C03619=1061.195,-112.854,-61.247,171.285,25.780,154.842
C03620=1061.201,-112.604,-61.257,171.286,25.781,154.842
C03621=1061.207,-112.354,-61.267,171.288,25.782,154.842
C03622=1061.214,-112.105,-61.276,171.290,25.783,154.842
C03623=1061.219,-111.855,-61.286,171.292,25.784,154.841
C03624=1061.225,-111.605,-61.296,171.294,25.785,154.842
C03625=1061.232,-111.356,-61.306,171.296,25.786,154.841
C03626=1061.237,-111.107,-61.315,171.297,25.787,154.841
C03627=1061.243,-110.857,-61.325,171.299,25.788,154.841
C03628=1061.250,-110.606,-61.335,171.301,25.789,154.841
C03629=1061.256,-110.356,-61.344,171.303,25.790,154.841
C03630=1061.263,-110.107,-61.354,171.304,25.790,154.841
C03631=1061.268,-109.892,-61.363,171.306,25.792,154.841
C03632=1061.273,-109.677,-61.371,171.308,25.792,154.841
C03633=1061.279,-109.462,-61.380,171.310,25.793,154.841
C03634=1061.284,-109.247,-61.388,171.311,25.794,154.841
C03635=1061.289,-109.032,-61.396,171.312,25.795,154.841
C03636=1061.295,-108.817,-61.405,171.314,25.795,154.841
C03637=1061.300,-108.602,-61.414,171.316,25.797,154.841
C03638=1061.305,-108.387,-61.421,171.318,25.797,154.841
C03639=1061.311,-108.138,-61.432,171.320,25.798,154.841
C03640=1061.317,-107.888,-61.441,171.321,25.800,154.841
C03641=1061.323,-107.638,-61.451,171.323,25.800,154.841
C03642=1061.329,-107.388,-61.461,171.325,25.801,154.841
C03643=1061.335,-107.139,-61.471,171.327,25.803,154.841
C03644=1061.342,-106.888,-61.481,171.329,25.803,154.841
C03645=1061.348,-106.638,-61.491,171.330,25.804,154.841
C03646=1061.354,-106.388,-61.501,171.332,25.806,154.841
C03647=1061.360,-106.139,-61.511,171.334,25.807,154.841
C03648=1061.366,-105.889,-61.521,171.336,25.807,154.841
C03649=1061.373,-105.640,-61.530,171.337,25.809,154.841
C03650=1061.378,-105.390,-61.541,171.339,25.810,154.841
C03651=1061.384,-105.140,-61.551,171.341,25.811,154.841
C03652=1061.391,-104.890,-61.560,171.343,25.812,154.841
C03653=1061.396,-104.641,-61.571,171.344,25.813,154.841
C03654=1061.403,-104.391,-61.581,171.346,25.814,154.841
C03655=1061.409,-104.141,-61.590,171.348,25.815,154.841
C03656=1061.415,-103.892,-61.601,171.350,25.816,154.841
C03657=1061.421,-103.642,-61.611,171.352,25.817,154.841
C03658=1061.427,-103.393,-61.621,171.354,25.818,154.841
C03659=1061.434,-103.142,-61.631,171.356,25.820,154.841
C03660=1061.439,-102.892,-61.641,171.358,25.821,154.841
C03661=1061.446,-102.643,-61.651,171.359,25.822,154.841
C03662=1061.452,-102.393,-61.661,171.361,25.823,154.841
C03663=1061.458,-102.144,-61.672,171.363,25.824,154.841
C03664=1061.464,-101.894,-61.681,171.365,25.825,154.841
C03665=1061.470,-101.644,-61.691,171.366,25.826,154.841
C03666=1061.476,-101.395,-61.702,171.368,25.827,154.841
C03667=1061.483,-101.144,-61.712,171.370,25.828,154.841
C03668=1061.489,-100.895,-61.722,171.372,25.830,154.841
C03669=1061.494,-100.645,-61.732,171.373,25.831,154.841
C03670=1061.501,-100.396,-61.743,171.375,25.831,154.841
C03671=1061.507,-100.146,-61.752,171.377,25.833,154.841
C03672=1061.513,-99.896,-61.763,171.379,25.834,154.841
C03673=1061.519,-99.647,-61.773,171.380,25.835,154.841
C03674=1061.526,-99.397,-61.783,171.383,25.836,154.841
C03675=1061.535,-99.043,-61.798,171.385,25.838,154.841
C03676=1061.543,-98.690,-61.812,171.387,25.840,154.841
C03677=1061.552,-98.335,-61.827,171.390,25.841,154.841
C03678=1061.560,-97.982,-61.841,171.393,25.843,154.841
C03679=1061.567,-97.732,-61.851,171.394,25.844,154.841
C03680=1061.573,-97.483,-61.861,171.396,25.845,154.841
C03681=1061.579,-97.233,-61.872,171.398,25.846,154.841
C03682=1061.585,-96.982,-61.882,171.400,25.847,154.841
C03683=1061.591,-96.733,-61.893,171.401,25.849,154.841
C03684=1061.597,-96.484,-61.904,171.404,25.851,154.841
C03685=1061.603,-96.234,-61.913,171.406,25.852,154.841
C03686=1061.609,-95.984,-61.924,171.407,25.853,154.841
C03687=1061.615,-95.735,-61.934,171.409,25.854,154.841
C03688=1061.621,-95.485,-61.944,171.411,25.855,154.841
C03689=1061.627,-95.235,-61.956,171.413,25.857,154.841
C03690=1061.633,-94.985,-61.965,171.414,25.858,154.841
C03691=1061.639,-94.736,-61.976,171.416,25.859,154.841
C03692=1061.646,-94.486,-61.986,171.418,25.861,154.841
C03693=1061.651,-94.236,-61.997,171.419,25.862,154.841
C03694=1061.658,-93.986,-62.007,171.421,25.863,154.841
C03695=1061.664,-93.737,-62.018,171.423,25.864,154.841
C03696=1061.669,-93.487,-62.028,171.425,25.865,154.841
C03697=1061.676,-93.238,-62.039,171.426,25.867,154.841
C03698=1061.681,-92.988,-62.049,171.428,25.868,154.841
C03699=1061.689,-92.738,-62.060,171.430,25.870,154.841
C03700=1061.694,-92.488,-62.070,171.431,25.871,154.841
C03701=1061.700,-92.239,-62.081,171.433,25.872,154.841
C03702=1061.706,-91.990,-62.091,171.435,25.873,154.841
C03703=1061.712,-91.739,-62.102,171.438,25.875,154.842
C03704=1061.719,-91.490,-62.112,171.439,25.876,154.842
C03705=1061.724,-91.240,-62.123,171.441,25.878,154.842
C03706=1061.730,-90.991,-62.134,171.443,25.879,154.842
C03707=1061.737,-90.741,-62.145,171.444,25.880,154.842
C03708=1061.743,-90.491,-62.155,171.446,25.882,154.842
C03709=1061.748,-90.241,-62.166,171.448,25.883,154.842
C03710=1061.755,-89.992,-62.176,171.450,25.884,154.842
C03711=1061.761,-89.742,-62.187,171.451,25.885,154.842
C03712=1061.767,-89.492,-62.198,171.453,25.887,154.842
C03713=1061.773,-89.242,-62.208,171.455,25.888,154.842
C03714=1061.779,-88.992,-62.219,171.456,25.889,154.842
C03715=1061.786,-88.743,-62.229,171.458,25.891,154.842
C03716=1061.792,-88.494,-62.240,171.460,25.892,154.842
C03717=1061.797,-88.244,-62.251,171.461,25.894,154.842
C03718=1061.805,-87.994,-62.262,171.463,25.895,154.842
C03719=1061.810,-87.744,-62.272,171.465,25.896,154.842
C03720=1061.816,-87.495,-62.283,171.467,25.898,154.842
C03721=1061.823,-87.245,-62.293,171.469,25.899,154.842
C03722=1061.829,-86.995,-62.304,171.471,25.900,154.842
C03723=1061.834,-86.746,-62.315,171.473,25.902,154.843
C03724=1061.841,-86.496,-62.326,171.474,25.903,154.843
C03725=1061.847,-86.246,-62.337,171.476,25.904,154.843
C03726=1061.853,-85.997,-62.347,171.478,25.906,154.843
C03727=1061.860,-85.747,-62.358,171.479,25.907,154.843
C03728=1061.865,-85.497,-62.368,171.481,25.909,154.843
C03729=1061.872,-85.247,-62.379,171.483,25.910,154.843
C03730=1061.878,-84.998,-62.390,171.484,25.912,154.843
C03731=1061.884,-84.748,-62.401,171.486,25.913,154.843
C03732=1061.890,-84.498,-62.412,171.488,25.914,154.843
C03733=1061.896,-84.248,-62.423,171.490,25.916,154.843
C03734=1061.902,-83.999,-62.433,171.491,25.917,154.843
C03735=1061.909,-83.749,-62.444,171.493,25.919,154.843
C03736=1061.915,-83.499,-62.455,171.495,25.920,154.843
C03737=1061.922,-83.250,-62.466,171.497,25.922,154.843
C03738=1061.927,-83.000,-62.477,171.499,25.923,154.843
C03739=1061.935,-82.718,-62.489,171.501,25.924,154.843
C03740=1061.942,-82.436,-62.501,171.502,25.926,154.844
C03741=1061.948,-82.154,-62.514,171.505,25.928,154.844
C03742=1061.955,-81.872,-62.526,171.507,25.929,154.844
C03743=1061.961,-81.622,-62.537,171.508,25.931,154.844
C03744=1061.968,-81.372,-62.548,171.510,25.932,154.844
C03745=1061.974,-81.123,-62.559,171.512,25.933,154.844
C03746=1061.980,-80.873,-62.570,171.513,25.935,154.844
C03747=1061.987,-80.624,-62.580,171.515,25.936,154.844
C03748=1061.993,-80.373,-62.591,171.517,25.938,154.844
C03749=1061.999,-80.124,-62.602,171.518,25.939,154.844
C03750=1062.005,-79.874,-62.614,171.520,25.941,154.844
C03751=1062.011,-79.625,-62.625,171.522,25.942,154.844
C03752=1062.018,-79.376,-62.635,171.523,25.944,154.844
C03753=1062.024,-79.125,-62.647,171.526,25.945,154.844
C03754=1062.030,-78.876,-62.657,171.528,25.947,154.845
C03755=1062.036,-78.626,-62.669,171.529,25.949,154.845
C03756=1062.042,-78.376,-62.680,171.531,25.950,154.845
C03757=1062.048,-78.127,-62.692,171.533,25.952,154.845
C03758=1062.054,-77.877,-62.702,171.534,25.953,154.845
C03759=1062.060,-77.628,-62.713,171.536,25.955,154.845
C03760=1062.066,-77.378,-62.725,171.538,25.957,154.845
C03761=1062.072,-77.128,-62.735,171.539,25.958,154.845
C03762=1062.078,-76.878,-62.747,171.541,25.960,154.845
C03763=1062.084,-76.629,-62.758,171.543,25.961,154.845
C03764=1062.091,-76.379,-62.769,171.544,25.962,154.845
C03765=1062.096,-76.129,-62.780,171.546,25.964,154.846
C03766=1062.103,-75.879,-62.792,171.548,25.965,154.846
C03767=1062.109,-75.630,-62.803,171.549,25.967,154.846
C03768=1062.115,-75.380,-62.814,171.551,25.969,154.846
C03769=1062.121,-75.131,-62.825,171.553,25.970,154.846
C03770=1062.127,-74.880,-62.837,171.554,25.972,154.846
C03771=1062.133,-74.632,-62.848,171.557,25.974,154.846
C03772=1062.140,-74.382,-62.859,171.558,25.975,154.846
C03773=1062.146,-74.132,-62.870,171.560,25.977,154.846
C03774=1062.152,-73.882,-62.881,171.562,25.979,154.846
C03775=1062.158,-73.633,-62.893,171.563,25.980,154.847
C03776=1062.164,-73.383,-62.904,171.565,25.982,154.847
C03777=1062.170,-73.133,-62.915,171.567,25.983,154.847
C03778=1062.177,-72.884,-62.927,171.568,25.985,154.847
C03779=1062.182,-72.634,-62.938,171.570,25.987,154.847
C03780=1062.187,-72.384,-62.950,171.572,25.989,154.847
C03781=1062.194,-72.135,-62.962,171.573,25.990,154.847
C03782=1062.200,-71.885,-62.972,171.575,25.992,154.847
C03783=1062.206,-71.635,-62.984,171.577,25.993,154.848
C03784=1062.212,-71.386,-62.995,171.578,25.995,154.848
C03785=1062.218,-71.136,-63.007,171.580,25.997,154.848
C03786=1062.224,-70.887,-63.019,171.581,25.999,154.848
C03787=1062.230,-70.637,-63.030,171.583,26.000,154.848
C03788=1062.236,-70.387,-63.041,171.585,26.002,154.848
C03789=1062.242,-70.137,-63.053,171.586,26.003,154.848
C03790=1062.247,-69.888,-63.064,171.588,26.005,154.848
C03791=1062.254,-69.638,-63.076,171.590,26.007,154.849
C03792=1062.260,-69.389,-63.087,171.592,26.009,154.849
C03793=1062.266,-69.139,-63.099,171.594,26.011,154.849
C03794=1062.272,-68.889,-63.111,171.595,26.012,154.849
C03795=1062.278,-68.639,-63.122,171.597,26.014,154.849
C03796=1062.284,-68.389,-63.134,171.599,26.016,154.849
C03797=1062.290,-68.140,-63.145,171.600,26.018,154.849
C03798=1062.296,-67.890,-63.157,171.602,26.019,154.849
C03799=1062.302,-67.641,-63.168,171.603,26.021,154.850
C03800=1062.308,-67.391,-63.180,171.605,26.022,154.850
C03801=1062.314,-67.142,-63.191,171.607,26.024,154.850
C03802=1062.320,-66.892,-63.203,171.608,26.026,154.850
C03803=1062.327,-66.612,-63.216,171.610,26.028,154.850
C03804=1062.334,-66.332,-63.229,171.612,26.030,154.850
C03805=1062.340,-66.052,-63.242,171.614,26.032,154.850
C03806=1062.347,-65.772,-63.255,171.616,26.034,154.851
C03807=1062.354,-65.523,-63.267,171.617,26.036,154.851
C03808=1062.360,-65.273,-63.278,171.619,26.037,154.851
C03809=1062.366,-65.023,-63.290,171.621,26.039,154.851
C03810=1062.372,-64.773,-63.302,171.622,26.041,154.851
C03811=1062.378,-64.524,-63.313,171.624,26.043,154.851
C03812=1062.384,-64.274,-63.326,171.625,26.044,154.851
C03813=1062.390,-64.024,-63.337,171.627,26.046,154.852
C03814=1062.396,-63.775,-63.349,171.629,26.048,154.852
C03815=1062.403,-63.525,-63.360,171.631,26.050,154.852
C03816=1062.408,-63.276,-63.372,171.633,26.052,154.852
C03817=1062.415,-63.026,-63.384,171.634,26.053,154.852
C03818=1062.421,-62.776,-63.395,171.636,26.055,154.852
C03819=1062.426,-62.527,-63.408,171.638,26.057,154.852
C03820=1062.433,-62.277,-63.419,171.639,26.059,154.852
C03821=1062.439,-62.027,-63.431,171.641,26.060,154.853
C03822=1062.445,-61.778,-63.442,171.643,26.062,154.853
C03823=1062.451,-61.529,-63.455,171.644,26.064,154.853
C03824=1062.458,-61.278,-63.466,171.646,26.066,154.853
C03825=1062.464,-61.029,-63.478,171.647,26.067,154.853
C03826=1062.470,-60.780,-63.490,171.649,26.069,154.853
C03827=1062.476,-60.529,-63.501,171.651,26.071,154.853
C03828=1062.483,-60.280,-63.513,171.652,26.073,154.854
C03829=1062.488,-60.031,-63.526,171.654,26.074,154.854
C03830=1062.494,-59.781,-63.538,171.656,26.076,154.854
C03831=1062.501,-59.531,-63.549,171.657,26.078,154.854
C03832=1062.506,-59.282,-63.561,171.659,26.080,154.854
C03833=1062.513,-59.032,-63.573,171.660,26.082,154.854
C03834=1062.519,-58.782,-63.584,171.662,26.084,154.855
C03835=1062.525,-58.532,-63.597,171.664,26.086,154.855
C03836=1062.531,-58.283,-63.608,171.665,26.087,154.855
C03837=1062.538,-58.034,-63.620,171.667,26.089,154.855
C03838=1062.544,-57.784,-63.633,171.669,26.091,154.855
C03839=1062.550,-57.534,-63.644,171.671,26.093,154.855
C03840=1062.556,-57.285,-63.656,171.673,26.095,154.855
C03841=1062.562,-57.035,-63.668,171.674,26.096,154.856
C03842=1062.569,-56.785,-63.680,171.676,26.098,154.856
C03843=1062.574,-56.535,-63.693,171.677,26.100,154.856
C03844=1062.581,-56.286,-63.705,171.679,26.102,154.856
C03845=1062.587,-56.036,-63.716,171.681,26.104,154.856
C03846=1062.593,-55.786,-63.728,171.682,26.106,154.856
C03847=1062.599,-55.537,-63.740,171.684,26.107,154.857
C03848=1062.606,-55.287,-63.752,171.685,26.109,154.857
C03849=1062.612,-55.037,-63.765,171.687,26.111,154.857
C03850=1062.618,-54.788,-63.776,171.689,26.113,154.857
C03851=1062.624,-54.539,-63.789,171.690,26.115,154.857
C03852=1062.630,-54.288,-63.800,171.692,26.117,154.857
C03853=1062.637,-54.039,-63.812,171.693,26.119,154.858
C03854=1062.643,-53.789,-63.825,171.695,26.120,154.858
C03855=1062.649,-53.540,-63.836,171.697,26.122,154.858
C03856=1062.656,-53.290,-63.848,171.698,26.124,154.858
C03857=1062.661,-53.041,-63.861,171.700,26.126,154.858
C03858=1062.668,-52.791,-63.873,171.701,26.128,154.858
C03859=1062.674,-52.541,-63.885,171.703,26.130,154.858
C03860=1062.681,-52.292,-63.897,171.705,26.131,154.859
C03861=1062.687,-52.042,-63.910,171.706,26.133,154.859
C03862=1062.693,-51.793,-63.921,171.708,26.135,154.859
C03863=1062.699,-51.543,-63.933,171.710,26.137,154.859
C03864=1062.705,-51.293,-63.946,171.711,26.139,154.859
C03865=1062.712,-51.044,-63.958,171.714,26.141,154.859
C03866=1062.718,-50.794,-63.970,171.715,26.143,154.860
C03867=1062.725,-50.516,-63.983,171.717,26.145,154.860
C03868=1062.732,-50.237,-63.997,171.718,26.147,154.860
C03869=1062.738,-49.958,-64.011,171.720,26.149,154.860
C03870=1062.745,-49.679,-64.025,171.722,26.151,154.860
C03871=1062.751,-49.430,-64.037,171.724,26.154,154.861
C03872=1062.757,-49.180,-64.049,171.726,26.155,154.861
C03873=1062.763,-48.930,-64.062,171.727,26.158,154.861
C03874=1062.769,-48.681,-64.074,171.729,26.159,154.861
C03875=1062.776,-48.432,-64.087,171.730,26.161,154.861
C03876=1062.782,-48.182,-64.099,171.732,26.164,154.862
C03877=1062.787,-47.933,-64.112,171.733,26.165,154.862
C03878=1062.794,-47.683,-64.123,171.735,26.168,154.862
C03879=1062.800,-47.433,-64.136,171.737,26.169,154.862
C03880=1062.806,-47.183,-64.149,171.738,26.172,154.862
C03881=1062.812,-46.933,-64.161,171.740,26.173,154.863
C03882=1062.818,-46.684,-64.173,171.741,26.175,154.863
C03883=1062.824,-46.435,-64.186,171.743,26.178,154.863
C03884=1062.830,-46.185,-64.199,171.744,26.179,154.863
C03885=1062.836,-45.935,-64.211,171.746,26.182,154.863
C03886=1062.842,-45.686,-64.223,171.748,26.183,154.863
C03887=1062.848,-45.436,-64.236,171.749,26.186,154.864
C03888=1062.854,-45.186,-64.248,171.751,26.187,154.864
C03889=1062.860,-44.937,-64.261,171.752,26.189,154.864
C03890=1062.867,-44.687,-64.273,171.754,26.191,154.864
C03891=1062.873,-44.437,-64.286,171.755,26.193,154.864
C03892=1062.879,-44.188,-64.299,171.757,26.196,154.865
C03893=1062.884,-43.938,-64.311,171.759,26.197,154.865
C03894=1062.891,-43.689,-64.323,171.760,26.200,154.865
C03895=1062.897,-43.440,-64.336,171.762,26.201,154.865
C03896=1062.903,-43.190,-64.348,171.763,26.204,154.866
C03897=1062.909,-42.940,-64.361,171.765,26.205,154.866
C03898=1062.916,-42.691,-64.374,171.766,26.208,154.866
C03899=1062.922,-42.441,-64.386,171.768,26.210,154.866
C03900=1062.928,-42.191,-64.399,171.770,26.212,154.866
C03901=1062.934,-41.942,-64.412,171.771,26.214,154.866
C03902=1062.940,-41.692,-64.424,171.773,26.216,154.867
C03903=1062.946,-41.442,-64.437,171.774,26.218,154.867
C03904=1062.953,-41.193,-64.450,171.776,26.220,154.867
C03905=1062.958,-40.943,-64.462,171.777,26.222,154.867
C03906=1062.964,-40.693,-64.475,171.779,26.224,154.868
C03907=1062.971,-40.444,-64.487,171.781,26.226,154.868
C03908=1062.977,-40.194,-64.500,171.782,26.228,154.868
C03909=1062.983,-39.945,-64.513,171.784,26.230,154.868
C03910=1062.989,-39.695,-64.526,171.785,26.232,154.868
C03911=1062.995,-39.445,-64.539,171.788,26.234,154.868
C03912=1063.002,-39.196,-64.551,171.789,26.237,154.869
C03913=1063.008,-38.947,-64.564,171.791,26.238,154.869
C03914=1063.014,-38.697,-64.576,171.792,26.241,154.869
C03915=1063.020,-38.447,-64.589,171.794,26.243,154.869
C03916=1063.026,-38.198,-64.602,171.796,26.245,154.870
C03917=1063.032,-37.948,-64.615,171.797,26.247,154.870
C03918=1063.038,-37.698,-64.628,171.799,26.249,154.870
C03919=1063.044,-37.449,-64.641,171.800,26.251,154.870
C03920=1063.050,-37.199,-64.654,171.802,26.253,154.871
C03921=1063.056,-36.949,-64.666,171.803,26.256,154.871
C03922=1063.062,-36.699,-64.679,171.805,26.257,154.871
C03923=1063.068,-36.450,-64.692,171.806,26.260,154.871
C03924=1063.074,-36.200,-64.705,171.808,26.262,154.871
C03925=1063.081,-35.951,-64.718,171.810,26.264,154.872
C03926=1063.086,-35.701,-64.731,171.811,26.266,154.872
C03927=1063.093,-35.452,-64.744,171.813,26.269,154.872
C03928=1063.099,-35.202,-64.756,171.814,26.270,154.872
C03929=1063.105,-34.953,-64.770,171.816,26.273,154.873
C03930=1063.111,-34.703,-64.782,171.817,26.275,154.873
C03931=1063.117,-34.425,-64.797,171.819,26.277,154.873
C03932=1063.124,-34.146,-64.812,171.820,26.280,154.873
C03933=1063.131,-33.869,-64.826,171.822,26.282,154.874
C03934=1063.138,-33.591,-64.840,171.824,26.284,154.874
C03935=1063.143,-33.341,-64.853,171.826,26.286,154.874
C03936=1063.150,-33.092,-64.866,171.827,26.289,154.874
C03937=1063.156,-32.842,-64.880,171.829,26.291,154.874
C03938=1063.162,-32.592,-64.892,171.830,26.293,154.875
C03939=1063.169,-32.342,-64.906,171.832,26.295,154.875
C03940=1063.174,-32.093,-64.918,171.834,26.297,154.875
C03941=1063.181,-31.843,-64.932,171.835,26.300,154.875
C03942=1063.187,-31.594,-64.945,171.837,26.302,154.876
C03943=1063.193,-31.344,-64.957,171.838,26.304,154.876
C03944=1063.199,-31.095,-64.971,171.840,26.306,154.876
C03945=1063.205,-30.846,-64.984,171.841,26.308,154.876
C03946=1063.210,-30.595,-64.997,171.843,26.310,154.877
C03947=1063.217,-30.346,-65.010,171.844,26.312,154.877
C03948=1063.223,-30.096,-65.023,171.846,26.315,154.877
C03949=1063.229,-29.846,-65.037,171.847,26.317,154.877
C03950=1063.236,-29.597,-65.050,171.849,26.319,154.877
C03951=1063.242,-29.348,-65.063,171.851,26.321,154.878
C03952=1063.248,-29.098,-65.076,171.852,26.323,154.878
C03953=1063.254,-28.849,-65.089,171.854,26.326,154.878
C03954=1063.260,-28.599,-65.102,171.855,26.327,154.878
C03955=1063.267,-28.349,-65.115,171.857,26.330,154.879
C03956=1063.273,-28.100,-65.128,171.858,26.332,154.879
C03957=1063.279,-27.850,-65.142,171.860,26.334,154.879
C03958=1063.285,-27.601,-65.155,171.861,26.337,154.879
C03959=1063.290,-27.351,-65.168,171.863,26.338,154.880
C03960=1063.297,-27.102,-65.181,171.864,26.341,154.880
C03961=1063.303,-26.852,-65.195,171.866,26.343,154.880
C03962=1063.310,-26.602,-65.208,171.867,26.345,154.880
C03963=1063.316,-26.352,-65.221,171.869,26.348,154.881
C03964=1063.321,-26.103,-65.235,171.870,26.350,154.881
C03965=1063.327,-25.854,-65.248,171.872,26.352,154.881
C03966=1063.333,-25.604,-65.261,171.874,26.354,154.881
C03967=1063.339,-25.355,-65.275,171.875,26.356,154.882
C03968=1063.345,-25.105,-65.288,171.877,26.359,154.882
C03969=1063.352,-24.855,-65.301,171.878,26.361,154.882
C03970=1063.357,-24.605,-65.315,171.880,26.363,154.882
C03971=1063.363,-24.356,-65.328,171.881,26.366,154.883
C03972=1063.370,-24.107,-65.342,171.882,26.368,154.883
C03973=1063.375,-23.857,-65.355,171.883,26.370,154.883
C03974=1063.381,-23.607,-65.368,171.885,26.372,154.884
C03975=1063.388,-23.357,-65.382,171.886,26.375,154.884
C03976=1063.393,-23.108,-65.396,171.888,26.377,154.884
C03977=1063.399,-22.859,-65.409,171.889,26.379,154.884
C03978=1063.406,-22.609,-65.422,171.891,26.382,154.885
C03979=1063.411,-22.360,-65.436,171.893,26.383,154.885
C03980=1063.418,-22.110,-65.450,171.894,26.386,154.885
C03981=1063.424,-21.860,-65.463,171.896,26.388,154.885
C03982=1063.430,-21.611,-65.477,171.897,26.390,154.886
C03983=1063.436,-21.362,-65.490,171.899,26.393,154.886
C03984=1063.442,-21.112,-65.503,171.900,26.395,154.886
C03985=1063.448,-20.862,-65.517,171.902,26.397,154.886
C03986=1063.454,-20.613,-65.531,171.903,26.399,154.887
C03987=1063.461,-20.364,-65.544,171.905,26.402,154.887
C03988=1063.466,-20.113,-65.557,171.906,26.404,154.887
C03989=1063.473,-19.863,-65.571,171.908,26.406,154.887
C03990=1063.479,-19.614,-65.584,171.909,26.409,154.888
C03991=1063.484,-19.365,-65.598,171.911,26.411,154.888
C03992=1063.491,-19.115,-65.611,171.912,26.413,154.888
C03993=1063.497,-18.865,-65.625,171.914,26.416,154.888
C03994=1063.503,-18.616,-65.639,171.915,26.418,154.889
C03995=1063.510,-18.337,-65.654,171.917,26.420,154.889
C03996=1063.516,-18.058,-65.669,171.919,26.423,154.889
C03997=1063.524,-17.779,-65.684,171.921,26.426,154.890
C03998=1063.530,-17.500,-65.700,171.922,26.428,154.890
C03999=1063.536,-17.250,-65.713,171.924,26.430,154.890
C04000=1063.543,-17.001,-65.727,171.925,26.433,154.890
C04001=1063.549,-16.752,-65.741,171.927,26.435,154.891
C04002=1063.555,-16.502,-65.755,171.928,26.437,154.891
C04003=1063.562,-16.252,-65.769,171.930,26.440,154.891
C04004=1063.567,-16.003,-65.782,171.931,26.442,154.892
C04005=1063.573,-15.754,-65.796,171.933,26.444,154.892
C04006=1063.580,-15.504,-65.809,171.935,26.447,154.892
C04007=1063.586,-15.254,-65.823,171.936,26.449,154.892
C04008=1063.592,-15.005,-65.836,171.938,26.451,154.893
C04009=1063.597,-14.755,-65.850,171.939,26.453,154.893
C04010=1063.604,-14.506,-65.865,171.941,26.456,154.893
C04011=1063.610,-14.256,-65.879,171.942,26.458,154.893
C04012=1063.615,-14.007,-65.892,171.944,26.460,154.894
C04013=1063.622,-13.757,-65.906,171.945,26.463,154.894
C04014=1063.628,-13.507,-65.920,171.947,26.466,154.894
C04015=1063.634,-13.258,-65.934,171.948,26.468,154.895
C04016=1063.640,-13.008,-65.948,171.950,26.470,154.895
C04017=1063.646,-12.759,-65.962,171.950,26.472,154.895
C04018=1063.652,-12.509,-65.975,171.952,26.475,154.895
C04019=1063.658,-12.259,-65.989,171.953,26.477,154.896
C04020=1063.664,-12.010,-66.004,171.955,26.479,154.896
C04021=1063.670,-11.761,-66.017,171.956,26.482,154.896
C04022=1063.676,-11.511,-66.032,171.958,26.484,154.897
C04023=1063.682,-11.261,-66.045,171.959,26.487,154.897
C04024=1063.688,-11.012,-66.059,171.961,26.489,154.897
C04025=1063.694,-10.762,-66.074,171.962,26.491,154.897
C04026=1063.700,-10.513,-66.087,171.964,26.494,154.898
C04027=1063.706,-10.264,-66.102,171.965,26.496,154.898
C04028=1063.712,-10.014,-66.116,171.967,26.499,154.898
C04029=1063.718,-9.764,-66.129,171.968,26.501,154.899
C04030=1063.724,-9.515,-66.143,171.970,26.503,154.899
C04031=1063.730,-9.265,-66.158,171.971,26.506,154.899
C04032=1063.737,-9.016,-66.171,171.973,26.508,154.899
C04033=1063.743,-8.766,-66.185,171.974,26.510,154.900
C04034=1063.749,-8.517,-66.199,171.976,26.513,154.900
C04035=1063.755,-8.267,-66.213,171.977,26.515,154.900
C04036=1063.761,-8.017,-66.227,171.979,26.518,154.901
C04037=1063.767,-7.768,-66.241,171.980,26.520,154.901
C04038=1063.773,-7.518,-66.256,171.982,26.522,154.901
C04039=1063.779,-7.269,-66.270,171.984,26.525,154.901
C04040=1063.785,-7.020,-66.283,171.985,26.527,154.902
C04041=1063.791,-6.770,-66.298,171.986,26.530,154.902
C04042=1063.797,-6.521,-66.312,171.988,26.532,154.902
C04043=1063.804,-6.271,-66.326,171.990,26.534,154.903
C04044=1063.810,-6.022,-66.340,171.990,26.537,154.903
C04045=1063.816,-5.771,-66.355,171.992,26.539,154.903
C04046=1063.821,-5.522,-66.369,171.993,26.541,154.903
C04047=1063.828,-5.273,-66.383,171.995,26.544,154.904
C04048=1063.834,-5.023,-66.397,171.996,26.546,154.904
C04049=1063.840,-4.773,-66.412,171.998,26.549,154.904
C04050=1063.846,-4.524,-66.425,171.999,26.551,154.905
C04051=1063.853,-4.274,-66.440,172.001,26.553,154.905
C04052=1063.858,-4.025,-66.454,172.002,26.556,154.905
C04053=1063.865,-3.776,-66.468,172.004,26.558,154.906
C04054=1063.871,-3.526,-66.482,172.005,26.561,154.906
C04055=1063.877,-3.277,-66.497,172.007,26.563,154.906
C04056=1063.883,-3.027,-66.511,172.008,26.565,154.906
C04057=1063.889,-2.778,-66.525,172.010,26.568,154.907
C04058=1063.895,-2.527,-66.540,172.011,26.570,154.907
C04059=1063.901,-2.248,-66.556,172.013,26.573,154.907
C04060=1063.908,-1.967,-66.571,172.014,26.576,154.908
C04061=1063.915,-1.686,-66.589,172.016,26.579,154.908
C04062=1063.921,-1.406,-66.605,172.018,26.582,154.908
C04063=1063.927,-1.156,-66.619,172.020,26.584,154.909
C04064=1063.933,-0.907,-66.633,172.021,26.587,154.909
C04065=1063.939,-0.656,-66.648,172.022,26.589,154.909
C04066=1063.945,-0.408,-66.662,172.023,26.591,154.910
C04067=1063.951,-0.158,-66.677,172.025,26.594,154.910
C04068=1063.957,0.092,-66.691,172.026,26.596,154.910
C04069=1063.963,0.341,-66.706,172.027,26.599,154.911
C04070=1063.969,0.590,-66.721,172.029,26.602,154.911
C04071=1063.975,0.840,-66.734,172.031,26.604,154.911
C04072=1063.981,1.090,-66.749,172.032,26.607,154.912
C04073=1063.987,1.339,-66.764,172.034,26.609,154.912
C04074=1063.993,1.589,-66.778,172.035,26.611,154.912
C04075=1063.999,1.838,-66.793,172.036,26.614,154.913
C04076=1064.005,2.087,-66.808,172.038,26.616,154.913
C04077=1064.011,2.338,-66.822,172.040,26.619,154.913
C04078=1064.017,2.587,-66.837,172.041,26.622,154.914
C04079=1064.023,2.836,-66.851,172.043,26.624,154.914
C04080=1064.029,3.086,-66.865,172.044,26.626,154.914
C04081=1064.035,3.336,-66.880,172.045,26.629,154.914
C04082=1064.041,3.584,-66.895,172.047,26.631,154.915
C04083=1064.047,3.834,-66.910,172.047,26.634,154.915
C04084=1064.053,4.084,-66.924,172.049,26.636,154.915
C04085=1064.059,4.333,-66.939,172.051,26.639,154.916
C04086=1064.065,4.582,-66.953,172.052,26.641,154.916
C04087=1064.071,4.832,-66.968,172.054,26.644,154.916
C04088=1064.077,5.082,-66.982,172.055,26.646,154.917
C04089=1064.083,5.331,-66.997,172.057,26.649,154.917
C04090=1064.089,5.581,-67.012,172.058,26.651,154.917
C04091=1064.095,5.830,-67.026,172.060,26.653,154.918
C04092=1064.102,6.079,-67.041,172.061,26.656,154.918
C04093=1064.107,6.329,-67.055,172.063,26.659,154.918
C04094=1064.113,6.579,-67.070,172.064,26.662,154.919
C04095=1064.120,6.828,-67.085,172.066,26.664,154.919
C04096=1064.126,7.077,-67.100,172.067,26.666,154.919
C04097=1064.132,7.327,-67.115,172.068,26.669,154.920
C04098=1064.138,7.576,-67.129,172.070,26.671,154.920
C04099=1064.144,7.826,-67.144,172.071,26.673,154.920
C04100=1064.150,8.076,-67.158,172.072,26.676,154.920
C04101=1064.156,8.325,-67.173,172.074,26.678,154.921
C04102=1064.162,8.574,-67.188,172.075,26.681,154.921
C04103=1064.169,8.824,-67.203,172.077,26.684,154.921
C04104=1064.174,9.073,-67.218,172.078,26.686,154.922
C04105=1064.180,9.323,-67.233,172.080,26.689,154.922
C04106=1064.186,9.572,-67.248,172.081,26.691,154.922
C04107=1064.192,9.822,-67.263,172.083,26.693,154.923
C04108=1064.199,10.072,-67.277,172.084,26.696,154.923
C04109=1064.204,10.321,-67.291,172.086,26.699,154.923
C04110=1064.211,10.571,-67.306,172.087,26.701,154.924
C04111=1064.217,10.820,-67.321,172.089,26.704,154.924
C04112=1064.223,11.070,-67.336,172.090,26.706,154.924
C04113=1064.229,11.319,-67.351,172.092,26.709,154.925
C04114=1064.236,11.569,-67.366,172.093,26.711,154.925
C04115=1064.242,11.818,-67.381,172.094,26.713,154.925
C04116=1064.247,12.067,-67.396,172.095,26.716,154.926
C04117=1064.253,12.317,-67.411,172.097,26.718,154.926
C04118=1064.260,12.567,-67.426,172.098,26.721,154.926
C04119=1064.266,12.816,-67.440,172.100,26.723,154.927
C04120=1064.272,13.065,-67.455,172.101,26.726,154.927
C04121=1064.278,13.315,-67.470,172.103,26.729,154.927
C04122=1064.285,13.565,-67.485,172.104,26.731,154.927
C04123=1064.292,13.847,-67.502,172.106,26.734,154.928
C04124=1064.299,14.130,-67.519,172.107,26.737,154.928
C04125=1064.305,14.412,-67.536,172.109,26.740,154.929
C04126=1064.312,14.694,-67.553,172.111,26.743,154.929
C04127=1064.318,14.944,-67.568,172.112,26.745,154.929
C04128=1064.324,15.194,-67.583,172.114,26.748,154.930
C04129=1064.330,15.442,-67.599,172.115,26.750,154.930
C04130=1064.336,15.692,-67.614,172.116,26.753,154.930
C04131=1064.342,15.942,-67.629,172.117,26.755,154.931
C04132=1064.348,16.192,-67.644,172.119,26.758,154.931
C04133=1064.354,16.440,-67.659,172.120,26.760,154.931
C04134=1064.360,16.690,-67.674,172.122,26.763,154.932
C04135=1064.366,16.940,-67.689,172.123,26.765,154.932
C04136=1064.372,17.188,-67.705,172.125,26.768,154.932
C04137=1064.378,17.438,-67.720,172.126,26.770,154.933
C04138=1064.384,17.688,-67.735,172.128,26.773,154.933
C04139=1064.391,17.938,-67.750,172.129,26.776,154.933
C04140=1064.396,18.187,-67.765,172.131,26.778,154.934
C04141=1064.402,18.437,-67.780,172.132,26.781,154.934
C04142=1064.409,18.686,-67.796,172.134,26.784,154.934
C04143=1064.414,18.936,-67.811,172.134,26.786,154.935
C04144=1064.420,19.185,-67.826,172.136,26.788,154.935
C04145=1064.426,19.434,-67.841,172.137,26.791,154.935
C04146=1064.432,19.684,-67.857,172.139,26.794,154.936
C04147=1064.439,19.933,-67.872,172.140,26.796,154.936
C04148=1064.445,20.183,-67.887,172.142,26.799,154.936
C04149=1064.450,20.432,-67.902,172.143,26.801,154.937
C04150=1064.457,20.681,-67.918,172.145,26.804,154.937
C04151=1064.463,20.931,-67.933,172.146,26.806,154.937
C04152=1064.469,21.181,-67.948,172.148,26.809,154.938
C04153=1064.474,21.430,-67.963,172.149,26.812,154.938
C04154=1064.481,21.679,-67.979,172.151,26.814,154.938
C04155=1064.486,21.929,-67.995,172.152,26.817,154.939
C04156=1064.493,22.179,-68.010,172.153,26.819,154.939
C04157=1064.498,22.427,-68.026,172.154,26.822,154.939
C04158=1064.504,22.677,-68.040,172.156,26.824,154.940
C04159=1064.510,22.927,-68.056,172.157,26.827,154.940
C04160=1064.517,23.176,-68.072,172.159,26.829,154.940
C04161=1064.522,23.426,-68.087,172.160,26.832,154.941
C04162=1064.528,23.675,-68.102,172.162,26.835,154.941
C04163=1064.534,23.924,-68.118,172.163,26.837,154.941
C04164=1064.541,24.174,-68.133,172.165,26.840,154.942
C04165=1064.547,24.423,-68.149,172.166,26.842,154.942
C04166=1064.553,24.673,-68.164,172.168,26.845,154.942
C04167=1064.559,24.923,-68.180,172.169,26.848,154.943
C04168=1064.565,25.171,-68.195,172.171,26.850,154.943
C04169=1064.570,25.421,-68.211,172.171,26.853,154.944
C04170=1064.577,25.670,-68.226,172.173,26.855,154.944
C04171=1064.583,25.920,-68.242,172.174,26.858,154.944
C04172=1064.589,26.169,-68.257,172.176,26.860,154.945
C04173=1064.595,26.419,-68.273,172.177,26.863,154.945
C04174=1064.601,26.669,-68.288,172.179,26.866,154.945
C04175=1064.607,26.918,-68.304,172.180,26.868,154.946
C04176=1064.613,27.167,-68.319,172.182,26.871,154.946
C04177=1064.619,27.417,-68.335,172.183,26.873,154.946
C04178=1064.625,27.666,-68.350,172.185,26.876,154.947
C04179=1064.631,27.916,-68.366,172.186,26.879,154.947
C04180=1064.637,28.166,-68.382,172.188,26.881,154.947
C04181=1064.644,28.415,-68.397,172.188,26.883,154.948
C04182=1064.649,28.665,-68.413,172.190,26.886,154.948
C04183=1064.655,28.913,-68.428,172.191,26.889,154.948
C04184=1064.661,29.163,-68.444,172.193,26.891,154.949
C04185=1064.667,29.412,-68.460,172.194,26.894,154.949
C04186=1064.673,29.662,-68.476,172.196,26.897,154.949
C04187=1064.680,29.946,-68.494,172.197,26.900,154.950
C04188=1064.687,30.229,-68.511,172.199,26.903,154.950
C04189=1064.694,30.513,-68.529,172.201,26.906,154.951
C04190=1064.700,30.797,-68.548,172.202,26.909,154.951
C04191=1064.707,31.047,-68.563,172.204,26.912,154.951
C04192=1064.713,31.296,-68.579,172.205,26.915,154.952
C04193=1064.718,31.545,-68.595,172.206,26.917,154.952
C04194=1064.724,31.795,-68.611,172.207,26.919,154.952
C04195=1064.730,32.044,-68.626,172.209,26.922,154.953
C04196=1064.736,32.294,-68.642,172.210,26.925,154.953
C04197=1064.742,32.543,-68.658,172.212,26.927,154.954
C04198=1064.748,32.793,-68.674,172.213,26.930,154.954
C04199=1064.754,33.042,-68.689,172.215,26.932,154.954
C04200=1064.760,33.292,-68.705,172.216,26.935,154.955
C04201=1064.766,33.541,-68.722,172.218,26.938,154.955
C04202=1064.772,33.791,-68.737,172.219,26.940,154.955
C04203=1064.778,34.040,-68.753,172.221,26.943,154.956
C04204=1064.784,34.289,-68.769,172.222,26.946,154.956
C04205=1064.790,34.539,-68.785,172.223,26.948,154.956
C04206=1064.796,34.789,-68.801,172.224,26.951,154.957
C04207=1064.803,35.038,-68.817,172.226,26.953,154.957
C04208=1064.809,35.287,-68.833,172.227,26.956,154.957
C04209=1064.814,35.536,-68.848,172.229,26.959,154.958
C04210=1064.820,35.786,-68.864,172.230,26.961,154.958
C04211=1064.826,36.035,-68.880,172.232,26.964,154.958
C04212=1064.832,36.284,-68.896,172.233,26.967,154.959
C04213=1064.838,36.533,-68.913,172.235,26.969,154.959
C04214=1064.844,36.783,-68.928,172.236,26.972,154.960
C04215=1064.850,37.033,-68.944,172.238,26.974,154.960
C04216=1064.857,37.282,-68.960,172.239,26.977,154.960
C04217=1064.862,37.531,-68.976,172.240,26.980,154.961
C04218=1064.868,37.780,-68.992,172.241,26.982,154.961
C04219=1064.874,38.030,-69.008,172.243,26.985,154.961
C04220=1064.880,38.280,-69.024,172.244,26.988,154.962
C04221=1064.886,38.529,-69.041,172.246,26.991,154.962
C04222=1064.892,38.778,-69.057,172.247,26.993,154.962
C04223=1064.898,39.028,-69.073,172.249,26.996,154.963
C04224=1064.904,39.277,-69.089,172.250,26.999,154.963
C04225=1064.909,39.527,-69.105,172.252,27.001,154.964
C04226=1064.915,39.776,-69.121,172.253,27.004,154.964
C04227=1064.921,40.026,-69.137,172.255,27.006,154.964
C04228=1064.928,40.275,-69.153,172.256,27.009,154.965
C04229=1064.934,40.524,-69.169,172.257,27.011,154.965
C04230=1064.940,40.774,-69.186,172.258,27.014,154.965
C04231=1064.946,41.023,-69.202,172.260,27.017,154.966
C04232=1064.952,41.272,-69.218,172.261,27.020,154.966
C04233=1064.958,41.522,-69.234,172.263,27.022,154.966
C04234=1064.964,41.771,-69.251,172.264,27.025,154.967
C04235=1064.970,42.021,-69.267,172.266,27.028,154.967
C04236=1064.976,42.270,-69.283,172.267,27.030,154.967
C04237=1064.982,42.520,-69.300,172.269,27.033,154.968
C04238=1064.988,42.769,-69.316,172.270,27.036,154.968
C04239=1064.994,43.018,-69.332,172.272,27.039,154.969
C04240=1065.000,43.268,-69.348,172.272,27.041,154.969
C04241=1065.006,43.517,-69.365,172.274,27.043,154.969
C04242=1065.012,43.766,-69.381,172.275,27.046,154.970
C04243=1065.017,44.016,-69.398,172.277,27.049,154.970
C04244=1065.023,44.265,-69.414,172.278,27.051,154.970
C04245=1065.029,44.515,-69.430,172.280,27.054,154.971
C04246=1065.035,44.764,-69.447,172.281,27.057,154.971
C04247=1065.041,45.013,-69.463,172.283,27.060,154.972
C04248=1065.046,45.263,-69.480,172.284,27.063,154.972
C04249=1065.052,45.512,-69.496,172.286,27.066,154.972
C04250=1065.058,45.762,-69.512,172.287,27.068,154.973
C04251=1065.065,46.046,-69.531,172.288,27.071,154.973
C04252=1065.071,46.330,-69.550,172.290,27.074,154.974
C04253=1065.078,46.614,-69.569,172.291,27.077,154.974
C04254=1065.085,46.898,-69.587,172.293,27.080,154.974
C04255=1065.091,47.147,-69.604,172.294,27.083,154.975
C04256=1065.097,47.396,-69.621,172.296,27.086,154.975
C04257=1065.103,47.645,-69.637,172.297,27.088,154.976
C04258=1065.109,47.895,-69.653,172.299,27.091,154.976
C04259=1065.114,48.144,-69.670,172.300,27.094,154.976
C04260=1065.120,48.394,-69.686,172.302,27.097,154.977
C04261=1065.126,48.642,-69.703,172.303,27.100,154.977
C04262=1065.132,48.892,-69.720,172.305,27.102,154.977
C04263=1065.137,49.141,-69.736,172.305,27.104,154.978
C04264=1065.144,49.392,-69.753,172.307,27.107,154.978
C04265=1065.150,49.641,-69.769,172.308,27.110,154.979
C04266=1065.156,49.890,-69.785,172.310,27.113,154.979
C04267=1065.161,50.139,-69.803,172.311,27.115,154.979
C04268=1065.167,50.389,-69.819,172.313,27.118,154.980
C04269=1065.173,50.638,-69.836,172.314,27.121,154.980
C04270=1065.179,50.887,-69.852,172.316,27.124,154.980
C04271=1065.184,51.136,-69.869,172.317,27.127,154.981
C04272=1065.191,51.386,-69.886,172.319,27.129,154.981
C04273=1065.197,51.636,-69.902,172.320,27.132,154.982
C04274=1065.203,51.885,-69.919,172.322,27.134,154.982
C04275=1065.208,52.134,-69.936,172.322,27.137,154.982
C04276=1065.214,52.383,-69.952,172.324,27.140,154.983
C04277=1065.220,52.633,-69.969,172.325,27.142,154.983
C04278=1065.226,52.883,-69.987,172.327,27.145,154.983
C04279=1065.232,53.132,-70.003,172.328,27.148,154.984
C04280=1065.238,53.381,-70.019,172.330,27.151,154.984
C04281=1065.245,53.630,-70.036,172.331,27.153,154.985
C04282=1065.250,53.880,-70.053,172.333,27.156,154.985
C04283=1065.256,54.130,-70.070,172.334,27.159,154.985
C04284=1065.263,54.378,-70.086,172.336,27.161,154.986
C04285=1065.268,54.628,-70.103,172.337,27.164,154.986
C04286=1065.274,54.877,-70.120,172.339,27.166,154.986
C04287=1065.280,55.126,-70.137,172.339,27.169,154.987
C04288=1065.286,55.377,-70.154,172.341,27.172,154.987
C04289=1065.292,55.625,-70.171,172.342,27.175,154.988
C04290=1065.298,55.875,-70.187,172.344,27.178,154.988
C04291=1065.304,56.124,-70.203,172.345,27.180,154.988
C04292=1065.310,56.374,-70.221,172.347,27.183,154.989
C04293=1065.316,56.623,-70.237,172.348,27.185,154.989
C04294=1065.322,56.872,-70.254,172.350,27.188,154.989
C04295=1065.328,57.121,-70.271,172.351,27.191,154.990
C04296=1065.334,57.371,-70.289,172.353,27.193,154.990
C04297=1065.340,57.620,-70.305,172.354,27.196,154.991
C04298=1065.346,57.870,-70.322,172.356,27.199,154.991
C04299=1065.352,58.119,-70.339,172.356,27.201,154.991
C04300=1065.358,58.369,-70.355,172.358,27.204,154.992
C04301=1065.364,58.618,-70.373,172.359,27.207,154.992
C04302=1065.370,58.867,-70.389,172.361,27.209,154.992
C04303=1065.377,59.116,-70.406,172.362,27.212,154.993
C04304=1065.382,59.366,-70.423,172.364,27.215,154.993
C04305=1065.388,59.615,-70.440,172.365,27.217,154.993
C04306=1065.393,59.865,-70.457,172.367,27.220,154.994
C04307=1065.400,60.114,-70.474,172.368,27.222,154.994
C04308=1065.406,60.363,-70.491,172.370,27.225,154.995
C04309=1065.412,60.612,-70.508,172.371,27.228,154.995
C04310=1065.419,60.862,-70.526,172.373,27.230,154.995
C04311=1065.425,61.111,-70.542,172.374,27.233,154.996
C04312=1065.430,61.360,-70.559,172.376,27.236,154.996
C04313=1065.437,61.610,-70.576,172.376,27.239,154.996
C04314=1065.443,61.859,-70.593,172.378,27.241,154.997
C04315=1065.450,62.143,-70.612,172.380,27.244,154.997
C04316=1065.457,62.426,-70.632,172.382,27.247,154.998
C04317=1065.463,62.710,-70.651,172.383,27.250,154.998
C04318=1065.470,62.993,-70.670,172.385,27.253,154.998
C04319=1065.476,63.243,-70.688,172.386,27.256,154.999
C04320=1065.482,63.492,-70.705,172.388,27.259,154.999
C04321=1065.488,63.742,-70.723,172.389,27.261,154.999
C04322=1065.495,63.991,-70.740,172.391,27.264,155.000
C04323=1065.501,64.240,-70.756,172.392,27.267,155.000
C04324=1065.507,64.490,-70.774,172.394,27.269,155.001
C04325=1065.513,64.739,-70.791,172.395,27.272,155.001
C04326=1065.518,64.988,-70.808,172.397,27.274,155.001
C04327=1065.524,65.238,-70.825,172.398,27.277,155.002
C04328=1065.531,65.487,-70.842,172.399,27.280,155.002
C04329=1065.536,65.736,-70.860,172.400,27.283,155.003
C04330=1065.543,65.986,-70.877,172.402,27.285,155.003
C04331=1065.548,66.235,-70.894,172.403,27.288,155.003
C04332=1065.554,66.485,-70.912,172.405,27.290,155.004
C04333=1065.560,66.734,-70.928,172.406,27.293,155.004
C04334=1065.566,66.983,-70.946,172.408,27.296,155.004
C04335=1065.572,67.233,-70.964,172.409,27.299,155.005
C04336=1065.578,67.481,-70.981,172.411,27.302,155.005
C04337=1065.584,67.730,-70.998,172.412,27.304,155.006
C04338=1065.589,67.981,-71.016,172.414,27.307,155.006
C04339=1065.596,68.230,-71.033,172.415,27.310,155.006
C04340=1065.602,68.479,-71.051,172.417,27.312,155.007
C04341=1065.607,68.728,-71.068,172.418,27.315,155.007
C04342=1065.614,68.977,-71.085,172.419,27.317,155.007
C04343=1065.620,69.227,-71.103,172.420,27.320,155.008
C04344=1065.625,69.476,-71.120,172.422,27.323,155.008
C04345=1065.632,69.726,-71.137,172.423,27.326,155.009
C04346=1065.637,69.975,-71.155,172.425,27.329,155.009
C04347=1065.643,70.224,-71.172,172.426,27.331,155.009
C04348=1065.649,70.474,-71.190,172.428,27.334,155.010
C04349=1065.655,70.722,-71.207,172.429,27.336,155.010
C04350=1065.661,70.972,-71.225,172.431,27.339,155.010
C04351=1065.667,71.221,-71.243,172.432,27.342,155.011
C04352=1065.672,71.471,-71.260,172.434,27.345,155.011
C04353=1065.678,71.721,-71.278,172.435,27.348,155.012
C04354=1065.684,71.969,-71.294,172.437,27.351,155.012
C04355=1065.691,72.219,-71.312,172.438,27.353,155.012
C04356=1065.696,72.468,-71.330,172.440,27.356,155.013
C04357=1065.702,72.717,-71.348,172.441,27.358,155.013
C04358=1065.708,72.967,-71.365,172.442,27.361,155.014
C04359=1065.714,73.216,-71.382,172.444,27.364,155.014
C04360=1065.720,73.465,-71.400,172.445,27.367,155.014
C04361=1065.726,73.714,-71.418,172.446,27.369,155.015
C04362=1065.732,73.964,-71.436,172.448,27.372,155.015
C04363=1065.737,74.213,-71.453,172.450,27.374,155.015
C04364=1065.743,74.463,-71.471,172.451,27.377,155.016
C04365=1065.750,74.712,-71.488,172.453,27.380,155.016
C04366=1065.755,74.961,-71.506,172.454,27.383,155.017
C04367=1065.761,75.210,-71.524,172.456,27.386,155.017
C04368=1065.767,75.460,-71.541,172.457,27.389,155.017
C04369=1065.773,75.709,-71.559,172.459,27.391,155.018
C04370=1065.778,75.958,-71.577,172.460,27.394,155.018
C04371=1065.784,76.208,-71.595,172.462,27.396,155.019
C04372=1065.791,76.457,-71.612,172.463,27.399,155.019
C04373=1065.797,76.706,-71.630,172.464,27.402,155.019
C04374=1065.803,76.955,-71.648,172.465,27.405,155.020
C04375=1065.809,77.205,-71.666,172.467,27.407,155.020
C04376=1065.814,77.454,-71.684,172.468,27.410,155.020
C04377=1065.820,77.703,-71.701,172.470,27.412,155.021
C04378=1065.826,77.953,-71.719,172.471,27.415,155.021
C04379=1065.834,78.236,-71.739,172.473,27.418,155.022
C04380=1065.840,78.520,-71.759,172.475,27.422,155.022
C04381=1065.846,78.803,-71.780,172.477,27.425,155.023
C04382=1065.853,79.086,-71.800,172.478,27.428,155.023
C04383=1065.859,79.336,-71.818,172.479,27.431,155.023
C04384=1065.864,79.585,-71.836,172.481,27.433,155.024
C04385=1065.870,79.835,-71.854,172.483,27.436,155.024
C04386=1065.876,80.083,-71.872,172.484,27.439,155.025
C04387=1065.882,80.333,-71.890,172.486,27.441,155.025
C04388=1065.888,80.582,-71.908,172.487,27.444,155.025
C04389=1065.894,80.832,-71.926,172.489,27.447,155.026
C04390=1065.900,81.080,-71.944,172.490,27.450,155.026
C04391=1065.906,81.330,-71.962,172.492,27.453,155.026
C04392=1065.911,81.579,-71.980,172.493,27.455,155.027
C04393=1065.917,81.829,-71.998,172.494,27.458,155.027
C04394=1065.923,82.077,-72.016,172.495,27.461,155.028
C04395=1065.929,82.327,-72.034,172.497,27.463,155.028
C04396=1065.935,82.577,-72.052,172.498,27.466,155.028
C04397=1065.940,82.826,-72.070,172.500,27.469,155.029
C04398=1065.947,83.075,-72.089,172.501,27.471,155.029
C04399=1065.952,83.324,-72.106,172.503,27.474,155.030
C04400=1065.958,83.574,-72.124,172.504,27.477,155.030
C04401=1065.964,83.823,-72.142,172.506,27.480,155.030
C04402=1065.970,84.072,-72.160,172.507,27.483,155.031
C04403=1065.976,84.321,-72.178,172.509,27.485,155.031
C04404=1065.982,84.571,-72.197,172.510,27.488,155.031
C04405=1065.988,84.820,-72.215,172.512,27.491,155.032
C04406=1065.993,85.070,-72.233,172.513,27.493,155.032
C04407=1066.000,85.319,-72.251,172.515,27.496,155.033
C04408=1066.005,85.568,-72.269,172.516,27.499,155.033
C04409=1066.012,85.817,-72.287,172.518,27.502,155.033
C04410=1066.018,86.067,-72.305,172.519,27.505,155.034
C04411=1066.022,86.316,-72.324,172.521,27.507,155.034
C04412=1066.029,86.565,-72.342,172.522,27.510,155.035
C04413=1066.035,86.815,-72.360,172.524,27.512,155.035
C04414=1066.041,87.063,-72.378,172.525,27.515,155.035
C04415=1066.047,87.313,-72.396,172.527,27.518,155.036
C04416=1066.053,87.561,-72.415,172.528,27.521,155.036
C04417=1066.058,87.811,-72.433,172.529,27.523,155.037
C04418=1066.065,88.061,-72.452,172.531,27.526,155.037
C04419=1066.070,88.310,-72.469,172.532,27.528,155.037
C04420=1066.076,88.559,-72.487,172.534,27.531,155.038
C04421=1066.083,88.808,-72.506,172.535,27.534,155.038
C04422=1066.088,89.057,-72.523,172.537,27.537,155.038
C04423=1066.094,89.307,-72.543,172.538,27.540,155.039
C04424=1066.100,89.557,-72.561,172.540,27.542,155.039
C04425=1066.106,89.805,-72.579,172.541,27.545,155.040
C04426=1066.112,90.054,-72.598,172.543,27.547,155.040
C04427=1066.118,90.304,-72.616,172.544,27.550,155.040
C04428=1066.124,90.553,-72.635,172.546,27.553,155.041
C04429=1066.130,90.802,-72.652,172.547,27.556,155.041
C04430=1066.136,91.052,-72.671,172.549,27.558,155.041
C04431=1066.141,91.302,-72.690,172.550,27.561,155.042
C04432=1066.147,91.550,-72.708,172.552,27.564,155.042
C04433=1066.153,91.800,-72.726,172.553,27.566,155.043
C04434=1066.159,92.049,-72.745,172.555,27.569,155.043
C04435=1066.165,92.298,-72.763,172.557,27.572,155.043
C04436=1066.170,92.548,-72.782,172.558,27.575,155.044
C04437=1066.177,92.797,-72.800,172.560,27.578,155.044
C04438=1066.182,93.045,-72.819,172.561,27.580,155.045
C04439=1066.188,93.295,-72.837,172.563,27.583,155.045
C04440=1066.194,93.544,-72.856,172.564,27.586,155.045
C04441=1066.199,93.793,-72.875,172.566,27.589,155.046
C04442=1066.205,94.043,-72.893,172.567,27.592,155.046
C04443=1066.212,94.325,-72.914,172.569,27.594,155.047
C04444=1066.219,94.609,-72.935,172.570,27.597,155.047
C04445=1066.225,94.893,-72.956,172.572,27.601,155.048
C04446=1066.232,95.177,-72.977,172.574,27.604,155.048
C04447=1066.238,95.426,-72.996,172.576,27.606,155.048
C04448=1066.243,95.675,-73.015,172.577,27.609,155.049
C04449=1066.250,95.924,-73.034,172.579,27.612,155.049
C04450=1066.256,96.174,-73.051,172.580,27.615,155.050
C04451=1066.261,96.423,-73.071,172.582,27.618,155.050
C04452=1066.267,96.672,-73.089,172.583,27.620,155.050
C04453=1066.273,96.921,-73.108,172.585,27.623,155.051
C04454=1066.279,97.171,-73.126,172.586,27.625,155.051
C04455=1066.285,97.420,-73.145,172.588,27.628,155.051
C04456=1066.291,97.669,-73.164,172.589,27.631,155.052
C04457=1066.296,97.918,-73.183,172.591,27.634,155.052
C04458=1066.303,98.167,-73.202,172.592,27.637,155.053
C04459=1066.308,98.417,-73.220,172.594,27.639,155.053
C04460=1066.315,98.666,-73.239,172.595,27.642,155.053
C04461=1066.320,98.915,-73.258,172.597,27.644,155.054
C04462=1066.326,99.164,-73.276,172.598,27.647,155.054
C04463=1066.332,99.414,-73.296,172.600,27.650,155.055
C04464=1066.338,99.663,-73.314,172.601,27.653,155.055
C04465=1066.344,99.912,-73.332,172.603,27.656,155.055
C04466=1066.349,100.161,-73.351,172.605,27.658,155.056
C04467=1066.356,100.410,-73.370,172.606,27.661,155.056
C04468=1066.361,100.660,-73.389,172.608,27.663,155.056
C04469=1066.368,100.909,-73.408,172.609,27.666,155.057
C04470=1066.374,101.158,-73.427,172.611,27.669,155.057
C04471=1066.379,101.407,-73.446,172.612,27.672,155.058
C04472=1066.385,101.656,-73.464,172.614,27.675,155.058
C04473=1066.391,101.906,-73.484,172.615,27.677,155.058
C04474=1066.396,102.155,-73.503,172.617,27.680,155.059
C04475=1066.403,102.404,-73.521,172.618,27.683,155.059
C04476=1066.408,102.653,-73.540,172.620,27.686,155.060
C04477=1066.414,102.902,-73.560,172.621,27.689,155.060
C04478=1066.419,103.152,-73.579,172.623,27.691,155.060
C04479=1066.426,103.401,-73.597,172.624,27.694,155.061
C04480=1066.431,103.650,-73.617,172.626,27.697,155.061
C04481=1066.437,103.899,-73.636,172.627,27.699,155.062
C04482=1066.443,104.148,-73.654,172.629,27.702,155.062
C04483=1066.449,104.398,-73.673,172.631,27.705,155.062
C04484=1066.454,104.647,-73.693,172.632,27.707,155.063
C04485=1066.460,104.896,-73.712,172.634,27.710,155.063
C04486=1066.466,105.146,-73.731,172.635,27.713,155.064
C04487=1066.472,105.394,-73.749,172.637,27.716,155.064
C04488=1066.477,105.644,-73.769,172.638,27.719,155.064
C04489=1066.483,105.893,-73.788,172.640,27.721,155.065
C04490=1066.489,106.142,-73.807,172.641,27.724,155.065
C04491=1066.495,106.392,-73.826,172.643,27.727,155.066
C04492=1066.501,106.641,-73.845,172.644,27.729,155.066
C04493=1066.507,106.890,-73.864,172.646,27.732,155.066
C04494=1066.513,107.139,-73.884,172.647,27.735,155.067
C04495=1066.518,107.388,-73.903,172.649,27.738,155.067
C04496=1066.524,107.637,-73.922,172.650,27.740,155.067
C04497=1066.530,107.886,-73.940,172.652,27.743,155.068
C04498=1066.536,108.136,-73.960,172.654,27.746,155.068
C04499=1066.542,108.385,-73.979,172.655,27.749,155.069
C04500=1066.548,108.634,-73.999,172.657,27.751,155.069
C04501=1066.553,108.883,-74.018,172.658,27.754,155.069
C04502=1066.560,109.133,-74.037,172.660,27.756,155.070
C04503=1066.566,109.382,-74.056,172.661,27.759,155.070
C04504=1066.571,109.631,-74.075,172.663,27.762,155.071
C04505=1066.577,109.880,-74.095,172.664,27.765,155.071
C04506=1066.584,110.129,-74.114,172.666,27.768,155.071
C04507=1066.590,110.412,-74.136,172.667,27.770,155.072
C04508=1066.596,110.697,-74.157,172.670,27.774,155.072
C04509=1066.603,110.980,-74.179,172.671,27.777,155.073
C04510=1066.610,111.264,-74.202,172.673,27.780,155.073
C04511=1066.615,111.513,-74.221,172.674,27.782,155.073
C04512=1066.621,111.762,-74.241,172.676,27.785,155.074
C04513=1066.627,112.011,-74.260,172.677,27.788,155.074
C04514=1066.633,112.260,-74.279,172.679,27.791,155.075
C04515=1066.639,112.509,-74.299,172.680,27.793,155.075
C04516=1066.645,112.759,-74.318,172.683,27.797,155.075
C04517=1066.651,113.008,-74.337,172.684,27.799,155.076
C04518=1066.657,113.257,-74.357,172.686,27.802,155.076
C04519=1066.663,113.506,-74.376,172.688,27.804,155.077
C04520=1066.668,113.756,-74.395,172.689,27.807,155.077
C04521=1066.674,114.005,-74.415,172.691,27.810,155.077
C04522=1066.680,114.254,-74.435,172.692,27.813,155.078
C04523=1066.686,114.503,-74.454,172.694,27.815,155.078
C04524=1066.691,114.752,-74.474,172.695,27.818,155.079
C04525=1066.697,115.001,-74.493,172.697,27.821,155.079
C04526=1066.703,115.250,-74.513,172.698,27.824,155.079
C04527=1066.708,115.499,-74.532,172.700,27.827,155.080
C04528=1066.714,115.748,-74.553,172.701,27.829,155.080
C04529=1066.719,115.998,-74.572,172.703,27.832,155.081
C04530=1066.725,116.247,-74.591,172.704,27.835,155.081
C04531=1066.731,116.496,-74.611,172.706,27.838,155.081
C04532=1066.737,116.745,-74.630,172.708,27.840,155.082
C04533=1066.743,116.994,-74.650,172.709,27.843,155.082
C04534=1066.748,117.244,-74.669,172.711,27.846,155.083
C04535=1066.754,117.493,-74.690,172.712,27.849,155.083
C04536=1066.759,117.742,-74.709,172.714,27.852,155.083
C04537=1066.765,117.991,-74.729,172.715,27.854,155.084
C04538=1066.771,118.240,-74.748,172.718,27.857,155.084
C04539=1066.777,118.489,-74.768,172.719,27.860,155.085
C04540=1066.783,118.739,-74.788,172.721,27.863,155.085
C04541=1066.788,118.988,-74.808,172.722,27.866,155.085
C04542=1066.794,119.237,-74.828,172.724,27.868,155.086
C04543=1066.800,119.486,-74.847,172.725,27.871,155.086
C04544=1066.806,119.735,-74.867,172.727,27.874,155.087
C04545=1066.811,119.984,-74.887,172.728,27.877,155.087
C04546=1066.817,120.233,-74.907,172.730,27.880,155.087
C04547=1066.822,120.483,-74.926,172.732,27.882,155.088
C04548=1066.828,120.732,-74.946,172.733,27.885,155.088
C04549=1066.834,120.981,-74.966,172.735,27.887,155.088
C04550=1066.840,121.230,-74.986,172.736,27.890,155.089
C04551=1066.845,121.479,-75.006,172.738,27.893,155.089
C04552=1066.851,121.728,-75.026,172.739,27.896,155.090
C04553=1066.857,121.978,-75.046,172.742,27.899,155.090
C04554=1066.863,122.227,-75.066,172.743,27.901,155.090
C04555=1066.869,122.476,-75.086,172.745,27.904,155.091
C04556=1066.874,122.725,-75.105,172.746,27.907,155.091
C04557=1066.880,122.974,-75.125,172.748,27.910,155.092
C04558=1066.886,123.223,-75.145,172.750,27.912,155.092
C04559=1066.892,123.472,-75.165,172.751,27.915,155.092
C04560=1066.898,123.721,-75.185,172.753,27.918,155.093
C04561=1066.903,123.970,-75.205,172.754,27.921,155.093
C04562=1066.909,124.219,-75.225,172.756,27.923,155.094
C04563=1066.916,124.469,-75.245,172.757,27.926,155.094
C04564=1066.922,124.718,-75.265,172.759,27.929,155.094
C04565=1066.927,124.967,-75.285,172.761,27.932,155.095
C04566=1066.933,125.216,-75.305,172.763,27.934,155.095
C04567=1066.939,125.466,-75.324,172.764,27.937,155.096
C04568=1066.945,125.714,-75.344,172.766,27.940,155.096
C04569=1066.950,125.963,-75.365,172.768,27.943,155.096
C04570=1066.956,126.213,-75.385,172.769,27.945,155.097
C04571=1066.963,126.497,-75.408,172.771,27.948,155.097
C04572=1066.970,126.780,-75.431,172.773,27.951,155.098
C04573=1066.976,127.063,-75.453,172.775,27.955,155.098
C04574=1066.983,127.346,-75.476,172.777,27.958,155.098
C04575=1066.988,127.595,-75.497,172.779,27.960,155.099
C04576=1066.994,127.844,-75.516,172.780,27.963,155.099
C04577=1067.000,128.094,-75.536,172.782,27.966,155.100
C04578=1067.007,128.343,-75.556,172.783,27.969,155.100
C04579=1067.012,128.592,-75.577,172.785,27.971,155.100
C04580=1067.018,128.841,-75.597,172.786,27.974,155.101
C04581=1067.024,129.090,-75.617,172.788,27.976,155.101
C04582=1067.030,129.340,-75.637,172.790,27.979,155.102
C04583=1067.036,129.589,-75.657,172.792,27.982,155.102
C04584=1067.042,129.837,-75.677,172.794,27.985,155.102
C04585=1067.048,130.086,-75.697,172.795,27.988,155.103
C04586=1067.054,130.336,-75.718,172.797,27.990,155.103
C04587=1067.060,130.585,-75.738,172.798,27.993,155.103
C04588=1067.066,130.834,-75.758,172.800,27.995,155.104
C04589=1067.071,131.083,-75.778,172.801,27.998,155.104
C04590=1067.077,131.333,-75.798,172.803,28.001,155.105
C04591=1067.083,131.582,-75.818,172.805,28.004,155.105
C04592=1067.088,131.831,-75.839,172.807,28.006,155.105
C04593=1067.094,132.080,-75.859,172.809,28.009,155.106
C04594=1067.100,132.330,-75.880,172.810,28.012,155.106
C04595=1067.107,132.578,-75.900,172.812,28.014,155.107
C04596=1067.112,132.827,-75.921,172.813,28.017,155.107
C04597=1067.118,133.076,-75.941,172.815,28.020,155.107
C04598=1067.123,133.325,-75.961,172.816,28.023,155.108
C04599=1067.130,133.574,-75.982,172.819,28.026,155.108
C04600=1067.135,133.823,-76.002,172.820,28.029,155.109
C04601=1067.141,134.072,-76.022,172.822,28.031,155.109
C04602=1067.146,134.321,-76.043,172.824,28.034,155.109
C04603=1067.152,134.571,-76.064,172.825,28.037,155.110
C04604=1067.158,134.820,-76.084,172.827,28.040,155.110
C04605=1067.163,135.069,-76.104,172.828,28.042,155.111
C04606=1067.170,135.317,-76.125,172.831,28.045,155.111
C04607=1067.175,135.567,-76.146,172.832,28.048,155.111
C04608=1067.181,135.816,-76.166,172.834,28.050,155.112
C04609=1067.187,136.065,-76.186,172.835,28.053,155.112
C04610=1067.193,136.315,-76.207,172.837,28.056,155.112
C04611=1067.199,136.564,-76.227,172.839,28.059,155.113
C04612=1067.204,136.812,-76.249,172.840,28.061,155.113
C04613=1067.210,137.061,-76.268,172.843,28.064,155.114
C04614=1067.216,137.311,-76.289,172.844,28.067,155.114
C04615=1067.222,137.560,-76.309,172.846,28.070,155.114
C04616=1067.227,137.809,-76.330,172.847,28.073,155.115
C04617=1067.233,138.058,-76.352,172.849,28.075,155.115
C04618=1067.239,138.307,-76.371,172.850,28.078,155.116
C04619=1067.245,138.556,-76.392,172.852,28.081,155.116
C04620=1067.251,138.805,-76.414,172.855,28.084,155.116
C04621=1067.257,139.054,-76.434,172.856,28.086,155.117
C04622=1067.262,139.303,-76.454,172.858,28.089,155.117
C04623=1067.268,139.553,-76.475,172.859,28.092,155.118
C04624=1067.274,139.801,-76.496,172.861,28.094,155.118
C04625=1067.279,140.050,-76.516,172.862,28.097,155.118
C04626=1067.285,140.300,-76.537,172.865,28.100,155.119
C04627=1067.291,140.549,-76.559,172.866,28.103,155.119
C04628=1067.297,140.797,-76.578,172.868,28.106,155.120
C04629=1067.303,141.047,-76.599,172.870,28.108,155.120
C04630=1067.308,141.296,-76.621,172.871,28.111,155.120
C04631=1067.314,141.545,-76.641,172.873,28.114,155.121
C04632=1067.320,141.794,-76.663,172.875,28.117,155.121
C04633=1067.326,142.043,-76.683,172.877,28.120,155.122
C04634=1067.331,142.292,-76.703,172.878,28.122,155.122
C04635=1067.338,142.575,-76.728,172.880,28.125,155.122
C04636=1067.344,142.859,-76.752,172.882,28.129,155.123
C04637=1067.351,143.142,-76.775,172.884,28.131,155.123
C04638=1067.357,143.425,-76.798,172.886,28.135,155.124
C04639=1067.363,143.674,-76.820,172.888,28.138,155.124
C04640=1067.368,143.923,-76.841,172.889,28.141,155.125
C04641=1067.375,144.173,-76.862,172.891,28.143,155.125
C04642=1067.380,144.422,-76.883,172.894,28.146,155.125
C04643=1067.386,144.670,-76.903,172.895,28.149,155.126
C04644=1067.392,144.920,-76.924,172.897,28.152,155.126
C04645=1067.398,145.168,-76.946,172.898,28.155,155.127
C04646=1067.403,145.418,-76.967,172.900,28.157,155.127
C04647=1067.409,145.667,-76.988,172.902,28.160,155.127
C04648=1067.415,145.916,-77.009,172.904,28.162,155.128
C04649=1067.421,146.165,-77.029,172.905,28.165,155.128
C04650=1067.426,146.414,-77.050,172.907,28.168,155.128
C04651=1067.433,146.663,-77.072,172.909,28.171,155.129
C04652=1067.438,146.911,-77.093,172.911,28.174,155.129
C04653=1067.444,147.161,-77.114,172.913,28.176,155.130
C04654=1067.450,147.410,-77.135,172.914,28.179,155.130
C04655=1067.455,147.660,-77.156,172.916,28.182,155.130
C04656=1067.461,147.908,-77.177,172.918,28.185,155.131
C04657=1067.467,148.157,-77.199,172.920,28.188,155.131
C04658=1067.473,148.406,-77.219,172.921,28.190,155.132
C04659=1067.479,148.655,-77.241,172.923,28.193,155.132
C04660=1067.485,148.904,-77.261,172.925,28.196,155.132
C04661=1067.491,149.154,-77.283,172.927,28.199,155.133
C04662=1067.496,149.402,-77.304,172.929,28.202,155.133
C04663=1067.501,149.651,-77.326,172.930,28.204,155.134
C04664=1067.507,149.901,-77.347,172.932,28.207,155.134
C04665=1067.513,150.149,-77.368,172.933,28.210,155.134
C04666=1067.519,150.399,-77.390,172.936,28.213,155.135
C04667=1067.524,150.648,-77.410,172.938,28.216,155.135
C04668=1067.530,150.897,-77.432,172.939,28.218,155.136
C04669=1067.536,151.145,-77.453,172.941,28.221,155.136
C04670=1067.542,151.395,-77.475,172.943,28.224,155.136
C04671=1067.547,151.644,-77.495,172.945,28.227,155.137
C04672=1067.553,151.893,-77.517,172.946,28.230,155.137
C04673=1067.559,152.141,-77.538,172.948,28.232,155.138
C04674=1067.565,152.391,-77.560,172.950,28.235,155.138
C04675=1067.571,152.639,-77.581,172.952,28.238,155.138
C04676=1067.576,152.889,-77.602,172.954,28.241,155.139
C04677=1067.581,153.138,-77.624,172.955,28.244,155.139
C04678=1067.587,153.387,-77.646,172.958,28.247,155.140
C04679=1067.593,153.635,-77.667,172.959,28.249,155.140
C04680=1067.599,153.885,-77.688,172.961,28.252,155.140
C04681=1067.605,154.134,-77.710,172.962,28.255,155.141
C04682=1067.611,154.383,-77.731,172.965,28.258,155.141
C04683=1067.617,154.632,-77.752,172.966,28.261,155.142
C04684=1067.622,154.881,-77.774,172.968,28.263,155.142
C04685=1067.628,155.130,-77.795,172.970,28.265,155.142
C04686=1067.633,155.379,-77.817,172.972,28.268,155.143
C04687=1067.639,155.628,-77.839,172.974,28.271,155.143
C04688=1067.645,155.876,-77.860,172.975,28.274,155.144
C04689=1067.651,156.126,-77.882,172.977,28.277,155.144
C04690=1067.657,156.375,-77.904,172.979,28.280,155.144
C04691=1067.662,156.624,-77.925,172.981,28.283,155.145
C04692=1067.668,156.873,-77.947,172.983,28.286,155.145
C04693=1067.674,157.121,-77.968,172.984,28.288,155.146
C04694=1067.679,157.371,-77.990,172.987,28.291,155.146
C04695=1067.685,157.619,-78.011,172.988,28.294,155.146
C04696=1067.691,157.869,-78.033,172.990,28.297,155.147
C04697=1067.697,158.118,-78.055,172.991,28.300,155.147
C04698=1067.702,158.367,-78.077,172.994,28.303,155.148
C04699=1067.709,158.650,-78.101,172.995,28.305,155.148
C04700=1067.715,158.933,-78.126,172.998,28.309,155.149
C04701=1067.722,159.216,-78.150,173.000,28.312,155.149
C04702=1067.729,159.499,-78.175,173.002,28.315,155.150
C04703=1067.734,159.748,-78.197,173.004,28.318,155.150
C04704=1067.740,159.997,-78.218,173.006,28.321,155.150
C04705=1067.746,160.246,-78.240,173.008,28.324,155.151
C04706=1067.752,160.495,-78.262,173.009,28.326,155.151
C04707=1067.757,160.744,-78.283,173.012,28.329,155.151
C04708=1067.763,160.993,-78.306,173.013,28.332,155.152
C04709=1067.770,161.242,-78.327,173.015,28.335,155.152
C04710=1067.774,161.491,-78.349,173.016,28.338,155.153
C04711=1067.780,161.740,-78.371,173.019,28.341,155.153
C04712=1067.785,161.989,-78.393,173.021,28.343,155.154
C04713=1067.791,162.238,-78.415,173.022,28.347,155.154
C04714=1067.797,162.486,-78.437,173.025,28.350,155.154
C04715=1067.802,162.736,-78.459,173.026,28.352,155.155
C04716=1067.808,162.985,-78.481,173.028,28.355,155.155
C04717=1067.813,163.234,-78.503,173.030,28.358,155.156
C04718=1067.819,163.483,-78.526,173.032,28.361,155.156
C04719=1067.824,163.731,-78.547,173.033,28.364,155.157
C04720=1067.830,163.981,-78.569,173.035,28.367,155.157
C04721=1067.835,164.230,-78.591,173.038,28.370,155.157
C04722=1067.841,164.478,-78.613,173.039,28.372,155.158
C04723=1067.847,164.728,-78.636,173.041,28.375,155.158
C04724=1067.853,164.977,-78.657,173.043,28.378,155.159
C04725=1067.858,165.225,-78.680,173.045,28.381,155.159
C04726=1067.863,165.474,-78.702,173.046,28.384,155.159
C04727=1067.869,165.724,-78.724,173.049,28.387,155.160
C04728=1067.875,165.972,-78.746,173.050,28.390,155.160
C04729=1067.880,166.221,-78.768,173.052,28.393,155.161
C04730=1067.886,166.471,-78.790,173.055,28.396,155.161
C04731=1067.891,166.719,-78.813,173.056,28.398,155.161
C04732=1067.897,166.968,-78.835,173.058,28.402,155.162
C04733=1067.903,167.217,-78.857,173.060,28.405,155.162
C04734=1067.908,167.466,-78.879,173.062,28.407,155.163
C04735=1067.913,167.715,-78.901,173.063,28.410,155.163
C04736=1067.920,167.964,-78.924,173.066,28.413,155.164
C04737=1067.925,168.213,-78.946,173.068,28.416,155.164
C04738=1067.930,168.461,-78.969,173.069,28.419,155.164
C04739=1067.937,168.711,-78.990,173.072,28.422,155.165
C04740=1067.942,168.960,-79.013,173.073,28.425,155.165
C04741=1067.947,169.208,-79.035,173.075,28.427,155.166
C04742=1067.954,169.457,-79.057,173.077,28.430,155.166
C04743=1067.959,169.707,-79.080,173.079,28.433,155.167
C04744=1067.965,169.955,-79.102,173.080,28.436,155.167
C04745=1067.970,170.204,-79.124,173.083,28.439,155.167
C04746=1067.976,170.453,-79.147,173.085,28.442,155.168
C04747=1067.982,170.702,-79.169,173.086,28.445,155.168
C04748=1067.988,170.951,-79.191,173.089,28.448,155.169
C04749=1067.993,171.200,-79.214,173.090,28.451,155.169
C04750=1067.999,171.449,-79.236,173.093,28.454,155.169
C04751=1068.004,171.698,-79.258,173.094,28.456,155.170
C04752=1068.010,171.947,-79.281,173.096,28.459,155.170
C04753=1068.016,172.196,-79.304,173.099,28.462,155.171
C04754=1068.022,172.445,-79.326,173.100,28.465,155.171
C04755=1068.027,172.693,-79.348,173.102,28.468,155.172
C04756=1068.033,172.943,-79.370,173.104,28.471,155.172
C04757=1068.039,173.191,-79.393,173.106,28.474,155.172
C04758=1068.044,173.440,-79.416,173.108,28.477,155.173
C04759=1068.051,173.690,-79.438,173.110,28.479,155.173
C04760=1068.056,173.938,-79.461,173.112,28.482,155.174
C04761=1068.061,174.187,-79.483,173.114,28.485,155.174
C04762=1068.067,174.436,-79.505,173.116,28.488,155.174
C04763=1068.074,174.719,-79.531,173.118,28.491,155.175
C04764=1068.080,175.001,-79.556,173.121,28.495,155.175
C04765=1068.087,175.284,-79.582,173.122,28.498,155.176
C04766=1068.093,175.567,-79.608,173.125,28.501,155.176
C04767=1068.099,175.815,-79.630,173.126,28.504,155.177
C04768=1068.105,176.064,-79.653,173.129,28.507,155.177
C04769=1068.111,176.314,-79.675,173.130,28.509,155.177
C04770=1068.117,176.562,-79.698,173.133,28.512,155.178
C04771=1068.123,176.811,-79.721,173.134,28.516,155.178
C04772=1068.128,177.060,-79.744,173.136,28.518,155.179
C04773=1068.134,177.309,-79.767,173.139,28.521,155.179
C04774=1068.140,177.558,-79.788,173.140,28.524,155.180
C04775=1068.145,177.807,-79.811,173.143,28.527,155.180
C04776=1068.151,178.055,-79.834,173.144,28.530,155.180
C04777=1068.157,178.304,-79.857,173.147,28.533,155.181
C04778=1068.163,178.553,-79.880,173.149,28.535,155.181
C04779=1068.169,178.802,-79.902,173.150,28.538,155.182
C04780=1068.174,179.051,-79.924,173.153,28.541,155.182
C04781=1068.180,179.300,-79.947,173.154,28.544,155.182
C04782=1068.186,179.549,-79.970,173.157,28.547,155.183
C04783=1068.192,179.798,-79.993,173.158,28.550,155.183
C04784=1068.198,180.047,-80.016,173.161,28.553,155.184
C04785=1068.204,180.295,-80.039,173.163,28.556,155.184
C04786=1068.210,180.544,-80.062,173.164,28.558,155.185
C04787=1068.215,180.793,-80.085,173.167,28.561,155.185
C04788=1068.221,181.042,-80.107,173.168,28.564,155.185
C04789=1068.227,181.291,-80.130,173.171,28.567,155.186
C04790=1068.233,181.540,-80.153,173.172,28.570,155.186
C04791=1068.239,181.789,-80.176,173.175,28.573,155.187
C04792=1068.245,182.037,-80.199,173.177,28.575,155.187
C04793=1068.250,182.286,-80.222,173.179,28.578,155.187
C04794=1068.257,182.536,-80.245,173.181,28.581,155.188
C04795=1068.262,182.785,-80.268,173.183,28.584,155.188
C04796=1068.269,183.033,-80.290,173.185,28.587,155.189
C04797=1068.275,183.282,-80.313,173.187,28.590,155.189
C04798=1068.280,183.531,-80.336,173.189,28.593,155.189
C04799=1068.286,183.780,-80.359,173.191,28.596,155.190
C04800=1068.292,184.029,-80.382,173.193,28.599,155.190
C04801=1068.298,184.278,-80.405,173.195,28.601,155.191
C04802=1068.303,184.527,-80.428,173.197,28.604,155.191
C04803=1068.309,184.776,-80.451,173.199,28.607,155.191
C04804=1068.315,185.025,-80.474,173.201,28.610,155.192
C04805=1068.321,185.273,-80.497,173.203,28.613,155.192
C04806=1068.327,185.522,-80.520,173.206,28.616,155.193
C04807=1068.332,185.771,-80.544,173.207,28.619,155.193
C04808=1068.337,186.020,-80.567,173.210,28.622,155.194
C04809=1068.343,186.269,-80.590,173.211,28.625,155.194
C04810=1068.348,186.518,-80.613,173.214,28.629,155.195
C04811=1068.354,186.766,-80.637,173.215,28.631,155.195
C04812=1068.360,187.015,-80.660,173.218,28.634,155.195
C04813=1068.365,187.264,-80.683,173.219,28.638,155.196
C04814=1068.370,187.513,-80.706,173.222,28.641,155.196
C04815=1068.377,187.762,-80.730,173.224,28.643,155.197
C04816=1068.381,188.011,-80.754,173.226,28.647,155.197
C04817=1068.387,188.260,-80.777,173.228,28.649,155.198
C04818=1068.393,188.508,-80.800,173.230,28.652,155.198
C04819=1068.399,188.757,-80.823,173.232,28.656,155.199
C04820=1068.404,189.006,-80.847,173.234,28.659,155.199
C04821=1068.411,189.255,-80.871,173.236,28.661,155.199
C04822=1068.416,189.504,-80.894,173.238,28.665,155.200
C04823=1068.421,189.753,-80.917,173.240,28.668,155.200
C04824=1068.427,190.001,-80.941,173.243,28.670,155.201
C04825=1068.432,190.251,-80.964,173.244,28.674,155.201
C04826=1068.438,190.499,-80.987,173.247,28.677,155.202
C04827=1068.444,190.781,-81.014,173.249,28.680,155.202
C04828=1068.451,191.064,-81.041,173.251,28.683,155.203
C04829=1068.457,191.347,-81.068,173.253,28.687,155.203
C04830=1068.464,191.628,-81.094,173.256,28.690,155.204
C04831=1068.470,191.877,-81.118,173.258,28.693,155.204
C04832=1068.475,192.126,-81.141,173.260,28.696,155.204
C04833=1068.481,192.375,-81.164,173.262,28.700,155.205
C04834=1068.487,192.624,-81.188,173.264,28.702,155.205
C04835=1068.492,192.873,-81.212,173.267,28.705,155.206
C04836=1068.498,193.121,-81.236,173.268,28.708,155.206
C04837=1068.504,193.370,-81.259,173.271,28.711,155.207
C04838=1068.509,193.619,-81.283,173.272,28.714,155.207
C04839=1068.515,193.868,-81.306,173.275,28.718,155.208
C04840=1068.521,194.117,-81.330,173.277,28.721,155.208
C04841=1068.527,194.365,-81.354,173.279,28.723,155.208
C04842=1068.533,194.614,-81.377,173.282,28.727,155.209
C04843=1068.538,194.863,-81.401,173.283,28.729,155.209
C04844=1068.544,195.111,-81.424,173.286,28.732,155.210
C04845=1068.550,195.361,-81.449,173.287,28.736,155.210
C04846=1068.555,195.610,-81.472,173.290,28.739,155.211
C04847=1068.561,195.858,-81.496,173.291,28.741,155.211
C04848=1068.567,196.107,-81.520,173.294,28.745,155.212
C04849=1068.573,196.356,-81.543,173.297,28.748,155.212
C04850=1068.578,196.605,-81.567,173.298,28.751,155.212
C04851=1068.584,196.853,-81.591,173.301,28.754,155.213
C04852=1068.589,197.102,-81.614,173.302,28.757,155.213
C04853=1068.596,197.351,-81.638,173.305,28.760,155.214
C04854=1068.601,197.600,-81.663,173.306,28.763,155.214
C04855=1068.607,197.849,-81.686,173.309,28.766,155.215
C04856=1068.613,198.097,-81.709,173.311,28.769,155.215
C04857=1068.619,198.346,-81.734,173.313,28.772,155.215
C04858=1068.625,198.595,-81.758,173.316,28.775,155.216
C04859=1068.630,198.844,-81.781,173.317,28.778,155.216
C04860=1068.637,199.093,-81.805,173.320,28.781,155.217
C04861=1068.642,199.341,-81.829,173.322,28.784,155.217
C04862=1068.648,199.590,-81.853,173.324,28.787,155.218
C04863=1068.653,199.839,-81.877,173.327,28.790,155.218
C04864=1068.660,200.088,-81.901,173.328,28.793,155.219
C04865=1068.665,200.336,-81.925,173.331,28.796,155.219
C04866=1068.671,200.585,-81.949,173.333,28.799,155.219
C04867=1068.677,200.834,-81.973,173.335,28.802,155.220
C04868=1068.683,201.082,-81.997,173.337,28.805,155.220
C04869=1068.688,201.332,-82.021,173.340,28.808,155.221
C04870=1068.694,201.580,-82.044,173.342,28.811,155.221
C04871=1068.700,201.829,-82.069,173.344,28.814,155.222
C04872=1068.706,202.078,-82.093,173.346,28.817,155.222
C04873=1068.712,202.327,-82.117,173.348,28.821,155.223
C04874=1068.718,202.576,-82.141,173.351,28.824,155.223
C04875=1068.724,202.824,-82.165,173.352,28.827,155.223
C04876=1068.729,203.073,-82.190,173.355,28.830,155.224
C04877=1068.734,203.321,-82.214,173.357,28.833,155.224
C04878=1068.741,203.570,-82.238,173.359,28.836,155.225
C04879=1068.746,203.819,-82.262,173.362,28.839,155.225
C04880=1068.752,204.068,-82.287,173.364,28.842,155.226
C04881=1068.757,204.317,-82.311,173.366,28.846,155.226
C04882=1068.763,204.565,-82.335,173.368,28.848,155.227
C04883=1068.769,204.814,-82.359,173.370,28.852,155.227
C04884=1068.775,205.063,-82.383,173.372,28.855,155.228
C04885=1068.780,205.311,-82.408,173.375,28.858,155.228
C04886=1068.786,205.561,-82.432,173.377,28.861,155.228
C04887=1068.792,205.809,-82.456,173.379,28.864,155.229
C04888=1068.798,206.058,-82.481,173.382,28.867,155.229
C04889=1068.803,206.307,-82.505,173.383,28.870,155.230
C04890=1068.808,206.555,-82.529,173.386,28.873,155.230
C04891=1068.833,207.599,-82.631,173.530,28.947,155.234
C04892=1068.838,207.814,-82.653,173.531,28.950,155.234
C04893=1068.843,208.029,-82.674,173.533,28.953,155.235
C04894=1068.848,208.244,-82.697,173.535,28.957,155.236
C04895=1068.853,208.459,-82.718,173.537,28.961,155.236
C04896=1068.859,208.674,-82.740,173.538,28.964,155.237
C04897=1068.864,208.889,-82.761,173.540,28.968,155.237
C04898=1068.869,209.103,-82.784,173.541,28.971,155.238
C04899=1068.874,209.318,-82.805,173.543,28.975,155.238
C04900=1068.880,209.567,-82.830,173.545,28.979,155.239
C04901=1068.885,209.817,-82.856,173.548,28.983,155.240
C04902=1068.892,210.065,-82.881,173.549,28.987,155.241
C04903=1068.897,210.313,-82.906,173.552,28.991,155.241
C04904=1068.903,210.562,-82.931,173.553,28.995,155.242
C04905=1068.910,210.811,-82.957,173.556,28.999,155.242
C04906=1068.916,211.059,-82.982,173.557,29.003,155.243
C04907=1068.921,211.308,-83.008,173.559,29.007,155.244
C04908=1068.927,211.557,-83.032,173.561,29.011,155.245
C04909=1068.933,211.805,-83.058,173.563,29.015,155.245
C04910=1068.939,212.054,-83.083,173.566,29.019,155.246
C04911=1068.944,212.303,-83.109,173.567,29.023,155.247
C04912=1068.951,212.552,-83.134,173.570,29.027,155.247
C04913=1068.956,212.800,-83.159,173.571,29.031,155.248
C04914=1068.962,213.048,-83.184,173.574,29.035,155.249
C04915=1068.968,213.297,-83.210,173.575,29.039,155.249
C04916=1068.974,213.546,-83.236,173.578,29.043,155.250
C04917=1068.980,213.795,-83.261,173.580,29.047,155.251
C04918=1068.985,214.043,-83.287,173.582,29.052,155.251
C04919=1068.991,214.292,-83.312,173.584,29.056,155.252
C04920=1068.998,214.540,-83.337,173.586,29.059,155.253
C04921=1069.003,214.789,-83.363,173.588,29.063,155.253
C04922=1069.009,215.038,-83.389,173.589,29.068,155.254
C04923=1069.015,215.287,-83.415,173.592,29.072,155.255
C04924=1069.020,215.535,-83.439,173.594,29.076,155.255
C04925=1069.027,215.784,-83.465,173.596,29.079,155.256
C04926=1069.032,216.032,-83.491,173.598,29.084,155.257
C04927=1069.038,216.281,-83.517,173.600,29.088,155.257
C04928=1069.045,216.529,-83.542,173.602,29.092,155.258
C04929=1069.050,216.778,-83.568,173.605,29.096,155.259
C04930=1069.056,217.027,-83.593,173.606,29.100,155.259
C04931=1069.062,217.276,-83.619,173.609,29.104,155.260
C04932=1069.068,217.525,-83.645,173.610,29.108,155.261
C04933=1069.073,217.772,-83.671,173.613,29.112,155.261
C04934=1069.079,218.021,-83.696,173.615,29.116,155.262
C04935=1069.086,218.270,-83.722,173.617,29.120,155.263
C04936=1069.091,218.519,-83.748,173.619,29.124,155.263
C04937=1069.098,218.767,-83.774,173.621,29.128,155.264
C04938=1069.103,219.016,-83.800,173.623,29.132,155.265
C04939=1069.109,219.264,-83.825,173.626,29.136,155.265
C04940=1069.115,219.513,-83.851,173.627,29.140,155.266
C04941=1069.121,219.761,-83.877,173.630,29.144,155.267
C04942=1069.127,220.010,-83.902,173.631,29.147,155.267
C04943=1069.133,220.259,-83.928,173.634,29.152,155.268
C04944=1069.139,220.507,-83.954,173.636,29.156,155.269
C04945=1069.145,220.756,-83.980,173.638,29.160,155.269
C04946=1069.151,221.005,-84.005,173.640,29.164,155.270
C04947=1069.157,221.253,-84.032,173.643,29.168,155.271
C04948=1069.162,221.470,-84.054,173.644,29.171,155.271
C04949=1069.168,221.687,-84.077,173.646,29.175,155.272
C04950=1069.172,221.905,-84.100,173.647,29.178,155.272
C04951=1069.178,222.122,-84.123,173.650,29.182,155.273
C04952=1069.183,222.339,-84.145,173.651,29.185,155.274
C04953=1069.187,222.556,-84.168,173.653,29.189,155.274
C04954=1069.193,222.774,-84.191,173.655,29.192,155.275
C04955=1069.198,222.991,-84.213,173.657,29.196,155.275
C04956=1069.204,223.240,-84.239,173.659,29.200,155.276
C04957=1069.209,223.488,-84.266,173.661,29.204,155.277
C04958=1069.216,223.737,-84.291,173.663,29.208,155.277
C04959=1069.221,223.985,-84.318,173.666,29.212,155.278
C04960=1069.227,224.234,-84.344,173.667,29.216,155.279
C04961=1069.233,224.482,-84.370,173.670,29.220,155.279
C04962=1069.239,224.731,-84.396,173.671,29.224,155.280
C04963=1069.245,224.979,-84.423,173.674,29.228,155.281
C04964=1069.250,225.228,-84.449,173.676,29.232,155.281
C04965=1069.257,225.477,-84.475,173.678,29.235,155.282
C04966=1069.262,225.725,-84.501,173.680,29.240,155.283
C04967=1069.268,225.974,-84.527,173.683,29.244,155.283
C04968=1069.274,226.222,-84.553,173.684,29.248,155.284
C04969=1069.280,226.470,-84.580,173.687,29.252,155.285
C04970=1069.286,226.720,-84.606,173.689,29.256,155.285
C04971=1069.292,226.968,-84.633,173.691,29.259,155.286
C04972=1069.298,227.217,-84.658,173.693,29.263,155.287
C04973=1069.304,227.465,-84.685,173.696,29.267,155.287
C04974=1069.310,227.714,-84.711,173.697,29.272,155.288
C04975=1069.315,227.962,-84.738,173.700,29.276,155.289
C04976=1069.322,228.211,-84.763,173.702,29.280,155.289
C04977=1069.327,228.459,-84.790,173.704,29.283,155.290
C04978=1069.334,228.708,-84.817,173.706,29.287,155.291
C04979=1069.339,228.957,-84.843,173.709,29.291,155.291
C04980=1069.346,229.205,-84.869,173.711,29.295,155.292
C04981=1069.352,229.454,-84.896,173.713,29.299,155.293
C04982=1069.357,229.702,-84.922,173.715,29.303,155.293
C04983=1069.363,229.951,-84.948,173.718,29.307,155.294
C04984=1069.369,230.200,-84.975,173.719,29.311,155.295
C04985=1069.375,230.448,-85.002,173.722,29.315,155.295
C04986=1069.381,230.697,-85.029,173.724,29.319,155.296
C04987=1069.387,230.945,-85.055,173.726,29.323,155.297
C04988=1069.393,231.193,-85.081,173.729,29.327,155.297
C04989=1069.399,231.441,-85.108,173.731,29.331,155.298
C04990=1069.404,231.690,-85.134,173.733,29.335,155.299
C04991=1069.411,231.939,-85.161,173.735,29.339,155.299
C04992=1069.416,232.188,-85.188,173.738,29.343,155.300
C04993=1069.422,232.436,-85.214,173.740,29.347,155.301
C04994=1069.428,232.685,-85.241,173.742,29.351,155.301
C04995=1069.434,232.933,-85.267,173.744,29.355,155.302
C04996=1069.440,233.182,-85.294,173.747,29.359,155.303
C04997=1069.446,233.430,-85.321,173.748,29.363,155.303
C04998=1069.452,233.679,-85.348,173.751,29.367,155.304
C04999=1069.457,233.927,-85.374,173.753,29.371,155.305
C05000=1069.463,234.175,-85.401,173.756,29.375,155.305
C05001=1069.470,234.424,-85.428,173.757,29.379,155.306
C05002=1069.475,234.673,-85.455,173.760,29.383,155.307
C05003=1069.480,234.922,-85.482,173.762,29.387,155.307
C05004=1069.485,235.135,-85.505,173.764,29.390,155.308
C05005=1069.491,235.347,-85.528,173.765,29.393,155.308
C05006=1069.496,235.561,-85.551,173.768,29.397,155.309
C05007=1069.501,235.774,-85.574,173.770,29.401,155.310
C05008=1069.506,235.987,-85.597,173.771,29.404,155.310
C05009=1069.511,236.200,-85.620,173.774,29.407,155.311
C05010=1069.516,236.413,-85.643,173.775,29.410,155.311
C05011=1069.521,236.626,-85.667,173.777,29.414,155.312
C05012=1069.527,236.875,-85.694,173.779,29.418,155.313
C05013=1069.533,237.123,-85.720,173.782,29.422,155.313
C05014=1069.539,237.372,-85.747,173.784,29.426,155.314
C05015=1069.545,237.621,-85.774,173.786,29.430,155.315
C05016=1069.551,237.869,-85.802,173.789,29.434,155.315
C05017=1069.556,238.117,-85.828,173.791,29.438,155.316
C05018=1069.562,238.365,-85.855,173.794,29.442,155.317
C05019=1069.568,238.615,-85.882,173.795,29.446,155.317
C05020=1069.575,238.862,-85.909,173.798,29.450,155.318
C05021=1069.580,239.111,-85.936,173.800,29.454,155.319
C05022=1069.587,239.360,-85.963,173.803,29.458,155.319
C05023=1069.592,239.608,-85.990,173.805,29.462,155.320
C05024=1069.598,239.856,-86.018,173.807,29.465,155.321
C05025=1069.604,240.105,-86.045,173.809,29.469,155.321
C05026=1069.610,240.354,-86.071,173.812,29.473,155.322
C05027=1069.616,240.602,-86.100,173.814,29.477,155.322
C05028=1069.622,240.851,-86.126,173.816,29.482,155.323
C05029=1069.627,241.099,-86.153,173.818,29.485,155.324
C05030=1069.634,241.347,-86.181,173.821,29.489,155.325
C05031=1069.640,241.596,-86.207,173.823,29.493,155.325
C05032=1069.645,241.844,-86.235,173.826,29.497,155.326
C05033=1069.652,242.093,-86.262,173.828,29.501,155.326
C05034=1069.657,242.341,-86.289,173.830,29.505,155.327
C05035=1069.664,242.590,-86.317,173.833,29.509,155.328
C05036=1069.669,242.838,-86.344,173.835,29.513,155.328
C05037=1069.676,243.087,-86.372,173.837,29.517,155.329
C05038=1069.681,243.336,-86.399,173.839,29.521,155.330
C05039=1069.687,243.583,-86.426,173.842,29.525,155.330
C05040=1069.693,243.833,-86.454,173.844,29.529,155.331
C05041=1069.699,244.080,-86.481,173.847,29.533,155.332
C05042=1069.704,244.328,-86.509,173.848,29.537,155.332
C05043=1069.710,244.577,-86.536,173.851,29.541,155.333
C05044=1069.716,244.825,-86.564,173.853,29.545,155.334
C05045=1069.722,245.075,-86.591,173.856,29.549,155.335
C05046=1069.728,245.322,-86.619,173.858,29.553,155.335
C05047=1069.734,245.572,-86.646,173.860,29.557,155.336
C05048=1069.740,245.819,-86.674,173.863,29.561,155.336
C05049=1069.745,246.067,-86.702,173.865,29.565,155.337
C05050=1069.752,246.317,-86.729,173.868,29.568,155.338
C05051=1069.757,246.565,-86.757,173.870,29.572,155.338
C05052=1069.764,246.813,-86.784,173.873,29.577,155.339
C05053=1069.769,247.062,-86.812,173.874,29.581,155.340
C05054=1069.775,247.310,-86.839,173.877,29.585,155.340
C05055=1069.781,247.558,-86.867,173.879,29.588,155.341
C05056=1069.787,247.807,-86.896,173.882,29.592,155.342
C05057=1069.792,248.056,-86.923,173.884,29.597,155.343
C05058=1069.798,248.303,-86.950,173.886,29.601,155.343
C05059=1069.804,248.552,-86.978,173.888,29.605,155.344
C05060=1069.814,248.972,-87.025,173.893,29.612,155.345
C05061=1069.824,249.392,-87.072,173.897,29.618,155.346
C05062=1069.833,249.812,-87.120,173.901,29.625,155.347
C05063=1069.843,250.232,-87.167,173.904,29.632,155.348
C05064=1069.848,250.480,-87.195,173.907,29.636,155.349
C05065=1069.855,250.728,-87.222,173.909,29.639,155.350
C05066=1069.861,250.976,-87.250,173.912,29.644,155.350
C05067=1069.866,251.225,-87.279,173.915,29.648,155.351
C05068=1069.872,251.473,-87.307,173.917,29.652,155.352
C05069=1069.878,251.721,-87.334,173.919,29.655,155.352
C05070=1069.884,251.969,-87.362,173.921,29.659,155.353
C05071=1069.890,252.218,-87.391,173.924,29.664,155.354
C05072=1069.895,252.466,-87.419,173.926,29.668,155.355
C05073=1069.902,252.715,-87.446,173.929,29.672,155.355
C05074=1069.908,252.963,-87.475,173.931,29.676,155.356
C05075=1069.913,253.211,-87.503,173.934,29.680,155.356
C05076=1069.919,253.460,-87.531,173.936,29.683,155.357
C05077=1069.925,253.708,-87.558,173.938,29.687,155.358
C05078=1069.931,253.957,-87.587,173.941,29.692,155.359
C05079=1069.937,254.205,-87.615,173.943,29.696,155.359
C05080=1069.942,254.453,-87.643,173.946,29.700,155.360
C05081=1069.949,254.702,-87.671,173.948,29.703,155.360
C05082=1069.954,254.950,-87.699,173.951,29.707,155.361
C05083=1069.960,255.199,-87.727,173.953,29.711,155.362
C05084=1069.966,255.447,-87.755,173.956,29.715,155.362
C05085=1069.972,255.695,-87.784,173.957,29.719,155.363
C05086=1069.979,255.943,-87.812,173.960,29.723,155.364
C05087=1069.985,256.192,-87.840,173.963,29.727,155.365
C05088=1069.990,256.440,-87.868,173.965,29.731,155.365
C05089=1069.996,256.689,-87.896,173.968,29.735,155.366
C05090=1070.002,256.937,-87.925,173.970,29.739,155.366
C05091=1070.009,257.185,-87.953,173.973,29.743,155.367
C05092=1070.014,257.434,-87.981,173.975,29.747,155.368
C05093=1070.020,257.682,-88.009,173.978,29.751,155.368
C05094=1070.026,257.930,-88.038,173.981,29.755,155.369
C05095=1070.032,258.178,-88.066,173.983,29.759,155.370
C05096=1070.038,258.427,-88.094,173.985,29.763,155.371
C05097=1070.045,258.675,-88.123,173.987,29.767,155.371
C05098=1070.050,258.924,-88.151,173.990,29.771,155.372
C05099=1070.056,259.172,-88.179,173.992,29.775,155.372
C05100=1070.062,259.420,-88.208,173.995,29.778,155.373
C05101=1070.068,259.669,-88.237,173.997,29.782,155.374
C05102=1070.074,259.917,-88.265,174.000,29.786,155.374
C05103=1070.080,260.165,-88.293,174.003,29.790,155.375
C05104=1070.086,260.413,-88.321,174.005,29.794,155.376
C05105=1070.093,260.661,-88.350,174.008,29.798,155.376
C05106=1070.098,260.910,-88.379,174.010,29.802,155.377
C05107=1070.105,261.158,-88.408,174.013,29.806,155.378
C05108=1070.111,261.407,-88.436,174.015,29.810,155.378
C05109=1070.116,261.655,-88.464,174.018,29.814,155.379
C05110=1070.123,261.903,-88.493,174.021,29.818,155.380
C05111=1070.129,262.152,-88.521,174.022,29.822,155.380
C05112=1070.139,262.569,-88.569,174.026,29.828,155.381
C05113=1070.150,262.986,-88.618,174.031,29.835,155.383
C05114=1070.160,263.404,-88.666,174.035,29.841,155.384
C05115=1070.170,263.822,-88.714,174.039,29.848,155.385
C05116=1070.176,264.069,-88.743,174.042,29.852,155.386
C05117=1070.181,264.318,-88.771,174.044,29.856,155.386
C05118=1070.188,264.566,-88.800,174.047,29.860,155.387
C05119=1070.193,264.814,-88.830,174.050,29.864,155.387
C05120=1070.199,265.063,-88.858,174.052,29.868,155.388
C05121=1070.205,265.311,-88.887,174.055,29.872,155.389
C05122=1070.211,265.559,-88.916,174.057,29.876,155.390
C05123=1070.217,265.807,-88.945,174.060,29.880,155.390
C05124=1070.223,266.056,-88.974,174.062,29.884,155.391
C05125=1070.229,266.304,-89.003,174.065,29.888,155.391
C05126=1070.235,266.552,-89.032,174.068,29.892,155.392
C05127=1070.241,266.800,-89.061,174.070,29.896,155.393
C05128=1070.247,267.048,-89.089,174.073,29.900,155.394
C05129=1070.252,267.297,-89.119,174.075,29.904,155.394
C05130=1070.258,267.545,-89.148,174.078,29.908,155.395
C05131=1070.265,267.793,-89.177,174.080,29.912,155.396
C05132=1070.271,268.041,-89.206,174.083,29.916,155.396
C05133=1070.276,268.290,-89.235,174.086,29.920,155.397
C05134=1070.283,268.538,-89.264,174.088,29.924,155.398
C05135=1070.289,268.787,-89.293,174.091,29.928,155.398
C05136=1070.295,269.035,-89.322,174.093,29.932,155.399
C05137=1070.300,269.283,-89.351,174.096,29.936,155.400
C05138=1070.307,269.531,-89.380,174.099,29.940,155.400
C05139=1070.313,269.779,-89.409,174.101,29.944,155.401
C05140=1070.318,270.027,-89.439,174.104,29.948,155.402
C05141=1070.324,270.275,-89.468,174.106,29.952,155.402
C05142=1070.330,270.523,-89.497,174.109,29.956,155.403
C05143=1070.336,270.772,-89.526,174.111,29.960,155.404
C05144=1070.342,271.020,-89.555,174.114,29.964,155.404
C05145=1070.348,271.268,-89.585,174.117,29.968,155.405
C05146=1070.354,271.517,-89.614,174.119,29.972,155.406
C05147=1070.360,271.765,-89.643,174.122,29.976,155.406
C05148=1070.366,272.013,-89.673,174.124,29.980,155.407
C05149=1070.372,272.261,-89.703,174.127,29.984,155.408
C05150=1070.378,272.509,-89.732,174.130,29.988,155.409
C05151=1070.384,272.757,-89.761,174.132,29.992,155.409
C05152=1070.390,273.005,-89.790,174.135,29.996,155.410
C05153=1070.396,273.254,-89.820,174.137,30.000,155.411
C05154=1070.402,273.502,-89.849,174.140,30.004,155.411
C05155=1070.407,273.750,-89.879,174.142,30.008,155.412
C05156=1070.413,273.998,-89.909,174.145,30.012,155.413
C05157=1070.419,274.246,-89.938,174.148,30.016,155.413
C05158=1070.425,274.495,-89.968,174.151,30.020,155.414
C05159=1070.431,274.743,-89.997,174.154,30.024,155.415
C05160=1070.437,274.991,-90.027,174.156,30.029,155.415
C05161=1070.443,275.239,-90.056,174.159,30.033,155.416
C05162=1070.449,275.487,-90.086,174.162,30.037,155.417
C05163=1070.456,275.735,-90.116,174.164,30.040,155.417
C05164=1070.460,275.964,-90.143,174.167,30.044,155.418
C05165=1070.466,276.192,-90.170,174.168,30.048,155.419
C05166=1070.472,276.421,-90.197,174.171,30.052,155.419
C05167=1070.477,276.649,-90.225,174.174,30.056,155.420
C05168=1070.483,276.878,-90.252,174.176,30.059,155.421
C05169=1070.488,277.106,-90.279,174.179,30.063,155.421
C05170=1070.494,277.335,-90.307,174.182,30.067,155.422
C05171=1070.499,277.564,-90.334,174.183,30.070,155.423
C05172=1070.505,277.812,-90.364,174.186,30.074,155.423
C05173=1070.510,278.060,-90.394,174.189,30.079,155.424
C05174=1070.518,278.308,-90.424,174.192,30.083,155.425
C05175=1070.523,278.557,-90.453,174.195,30.087,155.425
C05176=1070.529,278.804,-90.484,174.197,30.091,155.426
C05177=1070.535,279.053,-90.513,174.200,30.095,155.427
C05178=1070.541,279.300,-90.543,174.202,30.099,155.427
C05179=1070.546,279.549,-90.573,174.205,30.103,155.428
C05180=1070.553,279.796,-90.603,174.207,30.107,155.429
C05181=1070.559,280.045,-90.633,174.210,30.111,155.429
C05182=1070.565,280.293,-90.663,174.213,30.115,155.430
C05183=1070.571,280.541,-90.693,174.215,30.119,155.431
C05184=1070.577,280.771,-90.720,174.218,30.123,155.432
C05185=1070.581,281.001,-90.748,174.221,30.127,155.432
C05186=1070.587,281.231,-90.776,174.223,30.131,155.433
C05187=1070.593,281.461,-90.804,174.226,30.135,155.434
C05188=1070.599,281.691,-90.832,174.228,30.138,155.434
C05189=1070.604,281.921,-90.859,174.231,30.142,155.435
C05190=1070.610,282.151,-90.888,174.234,30.146,155.435
C05191=1070.614,282.381,-90.916,174.235,30.149,155.436
C05192=1070.621,282.629,-90.946,174.239,30.154,155.437
C05193=1070.627,282.877,-90.976,174.241,30.158,155.437
C05194=1070.633,283.125,-91.006,174.244,30.162,155.438
C05195=1070.639,283.373,-91.036,174.247,30.166,155.439
C05196=1070.644,283.621,-91.066,174.249,30.170,155.440
C05197=1070.651,283.870,-91.097,174.252,30.174,155.440
C05198=1070.657,284.117,-91.128,174.254,30.178,155.441
C05199=1070.662,284.366,-91.157,174.257,30.182,155.442
C05200=1070.668,284.614,-91.188,174.261,30.187,155.442
C05201=1070.674,284.862,-91.218,174.263,30.191,155.443
C05202=1070.680,285.110,-91.249,174.266,30.195,155.444
C05203=1070.687,285.357,-91.278,174.268,30.199,155.445
C05204=1070.693,285.605,-91.309,174.271,30.203,155.445
C05205=1070.699,285.854,-91.339,174.274,30.207,155.446
C05206=1070.705,286.102,-91.370,174.276,30.211,155.447
C05207=1070.711,286.349,-91.400,174.280,30.215,155.447
C05208=1070.717,286.599,-91.430,174.282,30.220,155.448
C05209=1070.722,286.846,-91.460,174.285,30.224,155.449
C05210=1070.728,287.094,-91.491,174.288,30.227,155.449
C05211=1070.735,287.343,-91.522,174.290,30.232,155.450
C05212=1070.741,287.591,-91.552,174.293,30.236,155.451
C05213=1070.746,287.838,-91.582,174.296,30.240,155.452
C05214=1070.753,288.086,-91.614,174.299,30.244,155.452
C05215=1070.759,288.334,-91.644,174.302,30.248,155.453
C05216=1070.765,288.582,-91.674,174.304,30.252,155.454
C05217=1070.771,288.830,-91.705,174.307,30.256,155.454
C05218=1070.777,289.078,-91.735,174.310,30.261,155.455
C05219=1070.783,289.326,-91.766,174.313,30.265,155.456
C05220=1070.788,289.542,-91.792,174.315,30.268,155.457
C05221=1070.794,289.757,-91.819,174.317,30.272,155.457
C05222=1070.799,289.973,-91.845,174.320,30.276,155.458
C05223=1070.804,290.188,-91.872,174.323,30.279,155.458
C05224=1070.809,290.404,-91.899,174.325,30.283,155.459
C05225=1070.815,290.619,-91.926,174.327,30.287,155.460
C05226=1070.819,290.835,-91.953,174.330,30.290,155.460
C05227=1070.825,291.051,-91.980,174.332,30.294,155.461
C05228=1070.830,291.298,-92.010,174.335,30.298,155.462
C05229=1070.836,291.546,-92.041,174.338,30.302,155.462
C05230=1070.843,291.795,-92.071,174.340,30.306,155.463
C05231=1070.849,292.042,-92.102,174.344,30.310,155.464
C05232=1070.854,292.291,-92.134,174.346,30.315,155.465
C05233=1070.860,292.539,-92.164,174.349,30.319,155.465
C05234=1070.867,292.787,-92.196,174.352,30.323,155.466
C05235=1070.873,293.034,-92.226,174.354,30.327,155.467
C05236=1070.878,293.282,-92.257,174.358,30.331,155.467
C05237=1070.885,293.530,-92.288,174.361,30.336,155.468
C05238=1070.890,293.778,-92.319,174.363,30.340,155.469
C05239=1070.897,294.026,-92.350,174.366,30.344,155.470
C05240=1070.902,294.274,-92.381,174.369,30.348,155.470
C05241=1070.909,294.522,-92.412,174.372,30.352,155.471
C05242=1070.915,294.770,-92.443,174.375,30.357,155.472
C05243=1070.921,295.018,-92.473,174.377,30.361,155.473
C05244=1070.927,295.266,-92.505,174.381,30.365,155.473
C05245=1070.933,295.515,-92.536,174.383,30.369,155.474
C05246=1070.939,295.762,-92.567,174.386,30.373,155.475
C05247=1070.945,296.010,-92.599,174.389,30.378,155.476
C05248=1070.951,296.258,-92.629,174.392,30.382,155.476
C05249=1070.958,296.506,-92.661,174.395,30.386,155.477
C05250=1070.963,296.754,-92.692,174.398,30.390,155.478
C05251=1070.969,297.002,-92.723,174.400,30.394,155.478
C05252=1070.975,297.250,-92.754,174.404,30.399,155.479
C05253=1070.981,297.498,-92.786,174.406,30.403,155.480
C05254=1070.987,297.745,-92.817,174.409,30.408,155.481
C05255=1070.993,297.994,-92.848,174.412,30.411,155.481
C05256=1070.998,298.241,-92.880,174.415,30.416,155.482
C05257=1071.004,298.489,-92.912,174.418,30.420,155.483
C05258=1071.011,298.737,-92.943,174.420,30.425,155.484
C05259=1071.016,298.986,-92.974,174.423,30.429,155.485
C05260=1071.022,299.233,-93.005,174.427,30.434,155.485
C05261=1071.028,299.481,-93.037,174.429,30.437,155.486
C05262=1071.034,299.728,-93.069,174.432,30.442,155.487
C05263=1071.040,299.976,-93.100,174.435,30.446,155.488
C05264=1071.046,300.224,-93.131,174.438,30.451,155.488
C05265=1071.052,300.473,-93.163,174.441,30.455,155.489
C05266=1071.058,300.720,-93.194,174.443,30.459,155.490
C05267=1071.064,300.968,-93.226,174.447,30.464,155.491
C05268=1071.069,301.216,-93.258,174.450,30.468,155.491
C05269=1071.076,301.464,-93.289,174.452,30.472,155.492
C05270=1071.082,301.712,-93.321,174.455,30.476,155.493
C05271=1071.087,301.959,-93.353,174.459,30.481,155.494
C05272=1071.093,302.207,-93.385,174.461,30.485,155.494
C05273=1071.099,302.455,-93.416,174.464,30.490,155.495
C05274=1071.105,302.703,-93.448,174.467,30.494,155.496
C05275=1071.111,302.951,-93.480,174.470,30.498,155.497
C05276=1071.117,303.174,-93.508,174.473,30.502,155.497
C05277=1071.122,303.396,-93.536,174.475,30.506,155.498
C05278=1071.127,303.620,-93.565,174.478,30.510,155.499
C05279=1071.133,303.842,-93.594,174.481,30.514,155.499
C05280=1071.138,304.065,-93.622,174.483,30.518,155.500
C05281=1071.144,304.289,-93.651,174.486,30.522,155.501
C05282=1071.149,304.511,-93.679,174.489,30.526,155.502
C05283=1071.154,304.734,-93.708,174.491,30.529,155.502
C05284=1071.161,304.981,-93.740,174.494,30.534,155.503
C05285=1071.167,305.230,-93.772,174.498,30.538,155.504
C05286=1071.173,305.478,-93.804,174.500,30.543,155.505
C05287=1071.178,305.725,-93.836,174.503,30.547,155.505
C05288=1071.185,305.973,-93.867,174.506,30.552,155.506
C05289=1071.191,306.221,-93.900,174.509,30.556,155.507
C05290=1071.196,306.468,-93.931,174.512,30.560,155.508
C05291=1071.202,306.717,-93.963,174.515,30.564,155.508
C05292=1071.208,306.965,-93.995,174.518,30.569,155.509
C05293=1071.215,307.212,-94.028,174.521,30.573,155.510
C05294=1071.221,307.460,-94.060,174.524,30.577,155.511
C05295=1071.227,307.708,-94.091,174.527,30.582,155.512
C05296=1071.233,307.956,-94.123,174.531,30.586,155.512
C05297=1071.240,308.203,-94.155,174.533,30.591,155.513
C05298=1071.246,308.452,-94.188,174.536,30.595,155.514
C05299=1071.252,308.700,-94.220,174.539,30.599,155.515
C05300=1071.257,308.947,-94.252,174.542,30.604,155.515
C05301=1071.263,309.195,-94.284,174.545,30.608,155.516
C05302=1071.270,309.442,-94.317,174.548,30.613,155.517
C05303=1071.277,309.690,-94.348,174.551,30.617,155.518
C05304=1071.282,309.939,-94.380,174.555,30.621,155.519
C05305=1071.289,310.186,-94.413,174.557,30.626,155.519
C05306=1071.295,310.434,-94.445,174.560,30.630,155.520
C05307=1071.301,310.682,-94.478,174.563,30.635,155.521
C05308=1071.306,310.929,-94.509,174.566,30.639,155.522
C05309=1071.313,311.177,-94.541,174.570,30.643,155.523
C05310=1071.319,311.425,-94.573,174.572,30.648,155.523
C05311=1071.326,311.673,-94.606,174.575,30.652,155.524
C05312=1071.332,311.921,-94.638,174.579,30.657,155.525
C05313=1071.338,312.168,-94.671,174.581,30.661,155.526
C05314=1071.344,312.417,-94.703,174.585,30.665,155.526
C05315=1071.350,312.664,-94.736,174.588,30.670,155.527
C05316=1071.357,312.912,-94.769,174.591,30.674,155.528
C05317=1071.363,313.160,-94.800,174.594,30.679,155.529
C05318=1071.370,313.407,-94.833,174.597,30.683,155.530
C05319=1071.376,313.655,-94.865,174.600,30.687,155.530
C05320=1071.382,313.903,-94.897,174.603,30.692,155.531
C05321=1071.388,314.151,-94.930,174.606,30.696,155.532
C05322=1071.394,314.399,-94.962,174.609,30.701,155.533
C05323=1071.400,314.646,-94.995,174.613,30.705,155.533
C05324=1071.406,314.894,-95.028,174.615,30.710,155.534
C05325=1071.412,315.142,-95.061,174.618,30.714,155.535
C05326=1071.419,315.390,-95.094,174.622,30.719,155.536
C05327=1071.424,315.638,-95.126,174.624,30.724,155.537
C05328=1071.430,315.886,-95.159,174.628,30.728,155.538
C05329=1071.436,316.134,-95.192,174.631,30.733,155.539
C05330=1071.442,316.381,-95.225,174.634,30.737,155.539
C05331=1071.448,316.629,-95.258,174.637,30.742,155.540
C05332=1071.453,316.854,-95.288,174.640,30.746,155.541
C05333=1071.459,317.078,-95.318,174.642,30.750,155.542
C05334=1071.464,317.303,-95.347,174.645,30.754,155.542
C05335=1071.469,317.527,-95.377,174.648,30.758,155.543
C05336=1071.475,317.752,-95.407,174.651,30.763,155.544
C05337=1071.480,317.977,-95.437,174.654,30.767,155.545
C05338=1071.486,318.201,-95.467,174.657,30.771,155.545
C05339=1071.492,318.425,-95.497,174.659,30.775,155.546
C05340=1071.497,318.673,-95.530,174.662,30.780,155.547
C05341=1071.504,318.921,-95.563,174.666,30.785,155.548
C05342=1071.509,319.168,-95.596,174.668,30.789,155.549
C05343=1071.515,319.416,-95.629,174.672,30.794,155.550
C05344=1071.521,319.664,-95.662,174.675,30.798,155.550
C05345=1071.527,319.911,-95.695,174.678,30.803,155.551
C05346=1071.534,320.160,-95.728,174.681,30.808,155.552
C05347=1071.540,320.408,-95.761,174.684,30.813,155.553
C05348=1071.546,320.655,-95.794,174.687,30.817,155.554
C05349=1071.552,320.903,-95.828,174.691,30.822,155.555
C05350=1071.558,321.150,-95.861,174.693,30.826,155.555
C05351=1071.564,321.398,-95.894,174.697,30.831,155.556
C05352=1071.570,321.646,-95.927,174.700,30.836,155.557
C05353=1071.576,321.894,-95.960,174.703,30.841,155.558
C05354=1071.583,322.141,-95.994,174.706,30.845,155.559
C05355=1071.588,322.389,-96.027,174.710,30.850,155.560
C05356=1071.595,322.637,-96.060,174.712,30.854,155.561
C05357=1071.601,322.884,-96.094,174.716,30.859,155.561
C05358=1071.607,323.132,-96.127,174.719,30.863,155.562
C05359=1071.614,323.380,-96.160,174.722,30.868,155.563
C05360=1071.619,323.628,-96.193,174.725,30.873,155.564
C05361=1071.626,323.875,-96.227,174.729,30.878,155.565
C05362=1071.631,324.123,-96.260,174.731,30.883,155.566
C05363=1071.639,324.370,-96.294,174.735,30.887,155.567
C05364=1071.644,324.618,-96.327,174.739,30.892,155.567
C05365=1071.650,324.866,-96.361,174.741,30.896,155.568
C05366=1071.656,325.113,-96.394,174.745,30.901,155.569
C05367=1071.662,325.362,-96.428,174.748,30.906,155.570
C05368=1071.669,325.609,-96.461,174.751,30.911,155.571
C05369=1071.675,325.857,-96.495,174.754,30.915,155.572
C05370=1071.682,326.104,-96.529,174.758,30.920,155.573
C05371=1071.687,326.352,-96.562,174.760,30.925,155.573
C05372=1071.694,326.599,-96.595,174.764,30.930,155.574
C05373=1071.700,326.848,-96.629,174.767,30.934,155.575
C05374=1071.707,327.095,-96.662,174.770,30.939,155.576
C05375=1071.712,327.343,-96.696,174.774,30.944,155.577
C05376=1071.719,327.591,-96.730,174.776,30.948,155.578
C05377=1071.725,327.838,-96.764,174.780,30.953,155.579
C05378=1071.731,328.086,-96.797,174.783,30.958,155.580
C05379=1071.738,328.333,-96.831,174.786,30.963,155.580
C05380=1071.744,328.580,-96.865,174.790,30.968,155.581
C05381=1071.750,328.829,-96.899,174.793,30.972,155.582
C05382=1071.757,329.076,-96.932,174.796,30.977,155.583
C05383=1071.763,329.324,-96.966,174.799,30.982,155.584
C05384=1071.769,329.572,-96.999,174.803,30.987,155.585
C05385=1071.776,329.820,-97.034,174.806,30.992,155.586
C05386=1071.782,330.067,-97.068,174.809,30.996,155.587
C05387=1071.788,330.314,-97.101,174.813,31.001,155.587
C05388=1071.794,330.536,-97.132,174.815,31.005,155.588
C05389=1071.800,330.757,-97.162,174.818,31.009,155.589
C05390=1071.806,330.979,-97.192,174.822,31.014,155.590
C05391=1071.811,331.200,-97.223,174.825,31.018,155.591
C05392=1071.817,331.422,-97.253,174.827,31.022,155.591
C05393=1071.822,331.643,-97.283,174.830,31.027,155.592
C05394=1071.828,331.865,-97.314,174.834,31.032,155.593
C05395=1071.834,332.086,-97.345,174.836,31.036,155.594
C05396=1071.840,332.334,-97.379,174.839,31.041,155.595
C05397=1071.845,332.581,-97.413,174.843,31.046,155.596
C05398=1071.852,332.829,-97.447,174.846,31.051,155.597
C05399=1071.858,333.076,-97.481,174.849,31.055,155.598
C05400=1071.864,333.324,-97.516,174.853,31.060,155.599
C05401=1071.870,333.571,-97.550,174.856,31.065,155.599
C05402=1071.877,333.819,-97.584,174.859,31.070,155.600
C05403=1071.882,334.067,-97.618,174.863,31.075,155.601
C05404=1071.889,334.315,-97.653,174.866,31.080,155.602
C05405=1071.895,334.562,-97.687,174.869,31.085,155.603
C05406=1071.901,334.810,-97.721,174.873,31.090,155.604
C05407=1071.907,335.057,-97.755,174.876,31.095,155.605
C05408=1071.914,335.305,-97.790,174.879,31.100,155.606
C05409=1071.920,335.553,-97.825,174.883,31.105,155.607
C05410=1071.926,335.800,-97.859,174.886,31.110,155.608
C05411=1071.933,336.048,-97.893,174.889,31.115,155.609
C05412=1071.938,336.295,-97.927,174.893,31.120,155.610
C05413=1071.945,336.543,-97.962,174.896,31.125,155.611
C05414=1071.952,336.790,-97.997,174.899,31.130,155.612
C05415=1071.958,337.038,-98.031,174.903,31.135,155.612
C05416=1071.964,337.285,-98.066,174.906,31.140,155.613
C05417=1071.970,337.532,-98.100,174.910,31.145,155.614
C05418=1071.977,337.780,-98.134,174.913,31.150,155.615
C05419=1071.983,338.028,-98.170,174.917,31.155,155.616
C05420=1071.989,338.275,-98.204,174.920,31.161,155.617
C05421=1071.995,338.523,-98.239,174.923,31.165,155.618
C05422=1072.001,338.770,-98.273,174.927,31.171,155.619
C05423=1072.008,339.018,-98.308,174.930,31.176,155.620
C05424=1072.014,339.266,-98.344,174.933,31.181,155.621
C05425=1072.020,339.513,-98.378,174.937,31.186,155.622
C05426=1072.026,339.760,-98.413,174.940,31.191,155.623
C05427=1072.033,340.008,-98.447,174.944,31.197,155.624
C05428=1072.038,340.255,-98.483,174.947,31.201,155.625
C05429=1072.045,340.503,-98.517,174.950,31.207,155.626
C05430=1072.051,340.751,-98.552,174.954,31.212,155.627
C05431=1072.058,340.997,-98.587,174.958,31.217,155.628
C05432=1072.063,341.246,-98.622,174.960,31.222,155.629
C05433=1072.070,341.493,-98.657,174.964,31.227,155.630
C05434=1072.077,341.741,-98.691,174.968,31.232,155.631
C05435=1072.083,341.988,-98.726,174.971,31.238,155.632
C05436=1072.089,342.235,-98.762,174.974,31.243,155.633
C05437=1072.095,342.483,-98.796,174.978,31.248,155.634
C05438=1072.102,342.731,-98.832,174.981,31.253,155.635
C05439=1072.107,342.978,-98.867,174.985,31.259,155.636
C05440=1072.114,343.225,-98.902,174.989,31.264,155.637
C05441=1072.121,343.473,-98.936,174.992,31.269,155.638
C05442=1072.127,343.721,-98.972,174.995,31.274,155.639
C05443=1072.133,343.968,-99.007,174.999,31.280,155.640
